MoveL Offs(p0,16.160800000000002,133.0456, 0), v100, z5, tool0;
MoveL Offs(p0,15.9875,133.9125, 0), v100, z5, tool0;
MoveL Offs(p0,15.787200000000002,134.9144, 0), v100, z5, tool0;
MoveL Offs(p0,15.5641,136.0327, 0), v100, z5, tool0;
MoveL Offs(p0,15.322400000000002,137.24880000000002, 0), v100, z5, tool0;
MoveL Offs(p0,15.066300000000002,138.54410000000001, 0), v100, z5, tool0;
MoveL Offs(p0,14.8,139.9, 0), v100, z5, tool0;
MoveL Offs(p0,14.232200000000002,142.5875, 0), v100, z5, tool0;
MoveL Offs(p0,13.713600000000003,144.79200000000006, 0), v100, z5, tool0;
MoveL Offs(p0,13.2214,146.54649999999998, 0), v100, z5, tool0;
MoveL Offs(p0,12.732800000000001,147.88400000000001, 0), v100, z5, tool0;
MoveL Offs(p0,12.225,148.8375, 0), v100, z5, tool0;
MoveL Offs(p0,11.6752,149.44, 0), v100, z5, tool0;
MoveL Offs(p0,11.060599999999999,149.7245, 0), v100, z5, tool0;
MoveL Offs(p0,10.3584,149.72400000000002, 0), v100, z5, tool0;
MoveL Offs(p0,9.5458,149.4715, 0), v100, z5, tool0;
MoveL Offs(p0,8.6,149.0, 0), v100, z5, tool0;
MoveL Offs(p0,8.192600000000002,148.78480000000002, 0), v100, z5, tool0;
MoveL Offs(p0,7.812800000000001,148.56240000000005, 0), v100, z5, tool0;
MoveL Offs(p0,7.4642,148.3376, 0), v100, z5, tool0;
MoveL Offs(p0,7.1504,148.11520000000002, 0), v100, z5, tool0;
MoveL Offs(p0,6.875,147.9, 0), v100, z5, tool0;
MoveL Offs(p0,6.6415999999999995,147.6968, 0), v100, z5, tool0;
MoveL Offs(p0,6.453799999999999,147.51039999999998, 0), v100, z5, tool0;
MoveL Offs(p0,6.3152,147.34560000000002, 0), v100, z5, tool0;
MoveL Offs(p0,6.2294,147.2072, 0), v100, z5, tool0;
MoveL Offs(p0,6.2,147.1, 0), v100, z5, tool0;
MoveL Offs(p0,5.95,144.525, 0), v100, z5, tool0;
MoveL Offs(p0,5.8184,143.6008, 0), v100, z5, tool0;
MoveL Offs(p0,5.6652000000000005,142.57940000000002, 0), v100, z5, tool0;
MoveL Offs(p0,5.492800000000001,141.4776, 0), v100, z5, tool0;
MoveL Offs(p0,5.3036,140.31220000000002, 0), v100, z5, tool0;
MoveL Offs(p0,5.1,139.1, 0), v100, z5, tool0;
MoveL Offs(p0,4.8993,137.8322, 0), v100, z5, tool0;
MoveL Offs(p0,4.718400000000001,136.50560000000002, 0), v100, z5, tool0;
MoveL Offs(p0,4.559099999999999,135.14540000000002, 0), v100, z5, tool0;
MoveL Offs(p0,4.4232000000000005,133.7768, 0), v100, z5, tool0;
MoveL Offs(p0,4.3125,132.425, 0), v100, z5, tool0;
MoveL Offs(p0,4.2288,131.1152, 0), v100, z5, tool0;
MoveL Offs(p0,4.173900000000001,129.8726, 0), v100, z5, tool0;
MoveL Offs(p0,4.1496,128.72240000000002, 0), v100, z5, tool0;
MoveL Offs(p0,4.1577,127.68980000000002, 0), v100, z5, tool0;
MoveL Offs(p0,4.2,126.8, 0), v100, z5, tool0;
MoveL Offs(p0,3.9,123.2, 0), v100, z5, tool0;
MoveL Offs(p0,3.5788,124.12820000000002, 0), v100, z5, tool0;
MoveL Offs(p0,3.334400000000001,125.71760000000003, 0), v100, z5, tool0;
MoveL Offs(p0,3.1656000000000004,127.7954, 0), v100, z5, tool0;
MoveL Offs(p0,3.0712,130.18880000000001, 0), v100, z5, tool0;
MoveL Offs(p0,3.05,132.725, 0), v100, z5, tool0;
MoveL Offs(p0,3.1008,135.2312, 0), v100, z5, tool0;
MoveL Offs(p0,3.2224000000000004,137.5346, 0), v100, z5, tool0;
MoveL Offs(p0,3.4136,139.46240000000003, 0), v100, z5, tool0;
MoveL Offs(p0,3.6732,140.8418, 0), v100, z5, tool0;
MoveL Offs(p0,4.2624,141.74560000000002, 0), v100, z5, tool0;
MoveL Offs(p0,4.3636,141.91039999999998, 0), v100, z5, tool0;
MoveL Offs(p0,4.4432,142.0968, 0), v100, z5, tool0;
MoveL Offs(p0,4.5,142.3, 0), v100, z5, tool0;
MoveL Offs(p0,4.5328,142.5152, 0), v100, z5, tool0;
MoveL Offs(p0,4.5404,142.7376, 0), v100, z5, tool0;
MoveL Offs(p0,4.521600000000001,142.96240000000003, 0), v100, z5, tool0;
MoveL Offs(p0,4.4752,143.18480000000002, 0), v100, z5, tool0;
MoveL Offs(p0,4.4,143.4, 0), v100, z5, tool0;
MoveL Offs(p0,4.9022,146.56709999999998, 0), v100, z5, tool0;
MoveL Offs(p0,5.4144000000000005,148.1312, 0), v100, z5, tool0;
MoveL Offs(p0,6.025,149.7625, 0), v100, z5, tool0;
MoveL Offs(p0,6.6896,151.3488, 0), v100, z5, tool0;
MoveL Offs(p0,7.3638,152.7779, 0), v100, z5, tool0;
MoveL Offs(p0,8.003200000000001,153.93760000000003, 0), v100, z5, tool0;
MoveL Offs(p0,8.563400000000001,154.7157, 0), v100, z5, tool0;
MoveL Offs(p0,9.0,155.0, 0), v100, z5, tool0;
MoveL Offs(p0,9.431999999999999,155.2754, 0), v100, z5, tool0;
MoveL Offs(p0,9.632000000000001,155.4768, 0), v100, z5, tool0;
MoveL Offs(p0,9.85,155.725, 0), v100, z5, tool0;
MoveL Offs(p0,10.080000000000002,156.0152, 0), v100, z5, tool0;
MoveL Offs(p0,10.315999999999999,156.3426, 0), v100, z5, tool0;
MoveL Offs(p0,10.552000000000001,156.7024, 0), v100, z5, tool0;
MoveL Offs(p0,10.782,157.08980000000003, 0), v100, z5, tool0;
MoveL Offs(p0,11.0,157.5, 0), v100, z5, tool0;
MoveL Offs(p0,11.221,157.9102, 0), v100, z5, tool0;
MoveL Offs(p0,11.460000000000004,158.29760000000005, 0), v100, z5, tool0;
MoveL Offs(p0,11.711000000000002,158.6574, 0), v100, z5, tool0;
MoveL Offs(p0,11.968,158.98480000000004, 0), v100, z5, tool0;
MoveL Offs(p0,12.225,159.275, 0), v100, z5, tool0;
MoveL Offs(p0,12.475999999999999,159.5232, 0), v100, z5, tool0;
MoveL Offs(p0,12.715,159.7246, 0), v100, z5, tool0;
MoveL Offs(p0,12.936000000000002,159.8744, 0), v100, z5, tool0;
MoveL Offs(p0,13.133,159.96779999999998, 0), v100, z5, tool0;
MoveL Offs(p0,13.3,160.0, 0), v100, z5, tool0;
MoveL Offs(p0,14.082399999999998,160.29760000000002, 0), v100, z5, tool0;
MoveL Offs(p0,14.3125,160.45, 0), v100, z5, tool0;
MoveL Offs(p0,14.545599999999999,160.62640000000002, 0), v100, z5, tool0;
MoveL Offs(p0,14.7763,160.82319999999999, 0), v100, z5, tool0;
MoveL Offs(p0,14.999200000000002,161.0368, 0), v100, z5, tool0;
MoveL Offs(p0,15.2089,161.2636, 0), v100, z5, tool0;
MoveL Offs(p0,15.4,161.5, 0), v100, z5, tool0;
MoveL Offs(p0,15.943300000000004,162.06070000000003, 0), v100, z5, tool0;
MoveL Offs(p0,16.7584,162.64960000000005, 0), v100, z5, tool0;
MoveL Offs(p0,17.7931,163.24689999999998, 0), v100, z5, tool0;
MoveL Offs(p0,18.995200000000004,163.83280000000002, 0), v100, z5, tool0;
MoveL Offs(p0,20.3125,164.3875, 0), v100, z5, tool0;
MoveL Offs(p0,21.6928,164.8912, 0), v100, z5, tool0;
MoveL Offs(p0,23.0839,165.3241, 0), v100, z5, tool0;
MoveL Offs(p0,24.433600000000006,165.6664, 0), v100, z5, tool0;
MoveL Offs(p0,25.6897,165.8983, 0), v100, z5, tool0;
MoveL Offs(p0,26.8,166.0, 0), v100, z5, tool0;
MoveL Offs(p0,28.5088,165.70880000000002, 0), v100, z5, tool0;
MoveL Offs(p0,28.675,165.4875, 0), v100, z5, tool0;
MoveL Offs(p0,28.7512,165.17919999999998, 0), v100, z5, tool0;
MoveL Offs(p0,28.7446,164.7701, 0), v100, z5, tool0;
MoveL Offs(p0,28.6624,164.2464, 0), v100, z5, tool0;
MoveL Offs(p0,28.5118,163.5943, 0), v100, z5, tool0;
MoveL Offs(p0,28.3,162.8, 0), v100, z5, tool0;
MoveL Offs(p0,28.3,162.8, 0), v100, z5, tool0;
MoveJ Offs(p0,78.0,158.0, 10), v100, z1, tool0;
MoveL Offs(p0,77.6872,153.00560000000004, 0), v100, z5, tool0;
MoveL Offs(p0,77.32230000000001,149.8019, 0), v100, z5, tool0;
MoveL Offs(p0,76.8416,146.2688, 0), v100, z5, tool0;
MoveL Offs(p0,76.2625,142.5125, 0), v100, z5, tool0;
MoveL Offs(p0,75.60239999999999,138.6392, 0), v100, z5, tool0;
MoveL Offs(p0,74.87870000000001,134.7551, 0), v100, z5, tool0;
MoveL Offs(p0,74.1088,130.96640000000002, 0), v100, z5, tool0;
MoveL Offs(p0,73.3101,127.37930000000001, 0), v100, z5, tool0;
MoveL Offs(p0,72.5,124.1, 0), v100, z5, tool0;
MoveL Offs(p0,72.09270000000001,122.5702, 0), v100, z5, tool0;
MoveL Offs(p0,71.71360000000001,121.11360000000005, 0), v100, z5, tool0;
MoveL Offs(p0,71.3669,119.7494, 0), v100, z5, tool0;
MoveL Offs(p0,71.05680000000001,118.49680000000001, 0), v100, z5, tool0;
MoveL Offs(p0,70.7875,117.375, 0), v100, z5, tool0;
MoveL Offs(p0,70.5632,116.4032, 0), v100, z5, tool0;
MoveL Offs(p0,70.3881,115.60059999999999, 0), v100, z5, tool0;
MoveL Offs(p0,70.2664,114.9864, 0), v100, z5, tool0;
MoveL Offs(p0,70.20230000000001,114.5798, 0), v100, z5, tool0;
MoveL Offs(p0,70.2,114.4, 0), v100, z5, tool0;
MoveL Offs(p0,70.48960000000002,114.63760000000002, 0), v100, z5, tool0;
MoveL Offs(p0,70.7499,114.96339999999998, 0), v100, z5, tool0;
MoveL Offs(p0,71.0768,115.41280000000002, 0), v100, z5, tool0;
MoveL Offs(p0,71.4625,115.975, 0), v100, z5, tool0;
MoveL Offs(p0,71.8992,116.6392, 0), v100, z5, tool0;
MoveL Offs(p0,72.3791,117.3946, 0), v100, z5, tool0;
MoveL Offs(p0,72.89440000000002,118.2304, 0), v100, z5, tool0;
MoveL Offs(p0,73.43730000000001,119.13580000000002, 0), v100, z5, tool0;
MoveL Offs(p0,74.0,120.1, 0), v100, z5, tool0;
MoveL Offs(p0,75.3555,122.35350000000001, 0), v100, z5, tool0;
MoveL Offs(p0,76.48000000000003,123.95600000000005, 0), v100, z5, tool0;
MoveL Offs(p0,77.3705,124.9105, 0), v100, z5, tool0;
MoveL Offs(p0,78.024,125.22, 0), v100, z5, tool0;
MoveL Offs(p0,78.4375,124.8875, 0), v100, z5, tool0;
MoveL Offs(p0,78.60800000000002,123.91600000000001, 0), v100, z5, tool0;
MoveL Offs(p0,78.5325,122.30850000000001, 0), v100, z5, tool0;
MoveL Offs(p0,77.6315,117.19750000000002, 0), v100, z5, tool0;
MoveL Offs(p0,76.8,113.7, 0), v100, z5, tool0;
MoveL Offs(p0,75.96640000000001,110.50610000000002, 0), v100, z5, tool0;
MoveL Offs(p0,75.08720000000002,107.46880000000002, 0), v100, z5, tool0;
MoveL Offs(p0,74.16479999999999,104.59470000000002, 0), v100, z5, tool0;
MoveL Offs(p0,73.2016,101.8904, 0), v100, z5, tool0;
MoveL Offs(p0,72.2,99.3625, 0), v100, z5, tool0;
MoveL Offs(p0,71.1624,97.01759999999999, 0), v100, z5, tool0;
MoveL Offs(p0,70.0912,94.8623, 0), v100, z5, tool0;
MoveL Offs(p0,68.9888,92.9032, 0), v100, z5, tool0;
MoveL Offs(p0,67.8576,91.1469, 0), v100, z5, tool0;
MoveL Offs(p0,66.7,89.6, 0), v100, z5, tool0;
MoveL Offs(p0,64.4,86.7, 0), v100, z5, tool0;
MoveL Offs(p0,61.2,92.3, 0), v100, z5, tool0;
MoveL Offs(p0,60.6388,93.25610000000002, 0), v100, z5, tool0;
MoveL Offs(p0,59.9864,94.30880000000003, 0), v100, z5, tool0;
MoveL Offs(p0,59.2596,95.43469999999999, 0), v100, z5, tool0;
MoveL Offs(p0,58.475199999999994,96.6104, 0), v100, z5, tool0;
MoveL Offs(p0,57.65,97.8125, 0), v100, z5, tool0;
MoveL Offs(p0,56.8008,99.01759999999999, 0), v100, z5, tool0;
MoveL Offs(p0,55.944399999999995,100.2023, 0), v100, z5, tool0;
MoveL Offs(p0,55.097600000000014,101.3432, 0), v100, z5, tool0;
MoveL Offs(p0,54.27720000000001,102.41689999999998, 0), v100, z5, tool0;
MoveL Offs(p0,53.5,103.4, 0), v100, z5, tool0;
MoveL Offs(p0,49.0,109.0, 0), v100, z5, tool0;
MoveL Offs(p0,50.9,116.8, 0), v100, z5, tool0;
MoveL Offs(p0,51.2321,118.13260000000002, 0), v100, z5, tool0;
MoveL Offs(p0,51.56480000000001,119.58880000000006, 0), v100, z5, tool0;
MoveL Offs(p0,51.89269999999999,121.13619999999999, 0), v100, z5, tool0;
MoveL Offs(p0,52.21040000000001,122.74240000000002, 0), v100, z5, tool0;
MoveL Offs(p0,52.5125,124.375, 0), v100, z5, tool0;
MoveL Offs(p0,52.793600000000005,126.00160000000001, 0), v100, z5, tool0;
MoveL Offs(p0,53.0483,127.5898, 0), v100, z5, tool0;
MoveL Offs(p0,53.2712,129.1072, 0), v100, z5, tool0;
MoveL Offs(p0,53.4569,130.5214, 0), v100, z5, tool0;
MoveL Offs(p0,53.6,131.8, 0), v100, z5, tool0;
MoveL Offs(p0,53.82320000000002,134.04640000000003, 0), v100, z5, tool0;
MoveL Offs(p0,53.9618,135.0751, 0), v100, z5, tool0;
MoveL Offs(p0,54.113600000000005,136.0192, 0), v100, z5, tool0;
MoveL Offs(p0,54.275,136.8625, 0), v100, z5, tool0;
MoveL Offs(p0,54.4424,137.5888, 0), v100, z5, tool0;
MoveL Offs(p0,54.61220000000001,138.18189999999998, 0), v100, z5, tool0;
MoveL Offs(p0,54.7808,138.62560000000002, 0), v100, z5, tool0;
MoveL Offs(p0,54.9446,138.90370000000001, 0), v100, z5, tool0;
MoveL Offs(p0,55.1,139.0, 0), v100, z5, tool0;
MoveL Offs(p0,55.75040000000003,138.55440000000004, 0), v100, z5, tool0;
MoveL Offs(p0,56.057599999999994,138.03609999999998, 0), v100, z5, tool0;
MoveL Offs(p0,56.34320000000001,137.3552, 0), v100, z5, tool0;
MoveL Offs(p0,56.6,136.5375, 0), v100, z5, tool0;
MoveL Offs(p0,56.8208,135.6088, 0), v100, z5, tool0;
MoveL Offs(p0,56.998400000000004,134.5949, 0), v100, z5, tool0;
MoveL Offs(p0,57.125600000000006,133.5216, 0), v100, z5, tool0;
MoveL Offs(p0,57.1952,132.41469999999998, 0), v100, z5, tool0;
MoveL Offs(p0,57.2,131.3, 0), v100, z5, tool0;
MoveL Offs(p0,57.4403,128.0438, 0), v100, z5, tool0;
MoveL Offs(p0,57.5,128.0, 0), v100, z5, tool0;
MoveL Offs(p0,57.95980000000001,128.5038, 0), v100, z5, tool0;
MoveL Offs(p0,58.43040000000002,129.93040000000002, 0), v100, z5, tool0;
MoveL Offs(p0,58.8986,132.1526, 0), v100, z5, tool0;
MoveL Offs(p0,59.351200000000006,135.0432, 0), v100, z5, tool0;
MoveL Offs(p0,59.775,138.475, 0), v100, z5, tool0;
MoveL Offs(p0,60.15680000000001,142.32080000000002, 0), v100, z5, tool0;
MoveL Offs(p0,60.483399999999996,146.45340000000002, 0), v100, z5, tool0;
MoveL Offs(p0,60.74159999999999,150.74560000000002, 0), v100, z5, tool0;
MoveL Offs(p0,60.9182,155.07020000000003, 0), v100, z5, tool0;
MoveL Offs(p0,61.0,159.3, 0), v100, z5, tool0;
MoveL Offs(p0,61.2125,159.8, 0), v100, z5, tool0;
MoveL Offs(p0,61.30239999999999,159.8688, 0), v100, z5, tool0;
MoveL Offs(p0,61.4067,159.92440000000002, 0), v100, z5, tool0;
MoveL Offs(p0,61.524800000000006,159.9656, 0), v100, z5, tool0;
MoveL Offs(p0,61.6561,159.9912, 0), v100, z5, tool0;
MoveL Offs(p0,61.8,160.0, 0), v100, z5, tool0;
MoveL Offs(p0,62.2879,159.6761, 0), v100, z5, tool0;
MoveL Offs(p0,62.88320000000002,158.78880000000004, 0), v100, z5, tool0;
MoveL Offs(p0,63.54329999999999,157.4647, 0), v100, z5, tool0;
MoveL Offs(p0,64.22560000000001,155.8304, 0), v100, z5, tool0;
MoveL Offs(p0,64.8875,154.0125, 0), v100, z5, tool0;
MoveL Offs(p0,65.4864,152.1376, 0), v100, z5, tool0;
MoveL Offs(p0,65.97970000000001,150.3323, 0), v100, z5, tool0;
MoveL Offs(p0,66.32480000000001,148.7232, 0), v100, z5, tool0;
MoveL Offs(p0,66.47909999999999,147.4369, 0), v100, z5, tool0;
MoveL Offs(p0,66.4,146.6, 0), v100, z5, tool0;
MoveL Offs(p0,65.9839,145.41660000000002, 0), v100, z5, tool0;
MoveL Offs(p0,65.85520000000001,144.77680000000004, 0), v100, z5, tool0;
MoveL Offs(p0,65.9833,144.6362, 0), v100, z5, tool0;
MoveL Offs(p0,66.8875,145.675, 0), v100, z5, tool0;
MoveL Offs(p0,68.4517,148.1778, 0), v100, z5, tool0;
MoveL Offs(p0,69.4048,149.8672, 0), v100, z5, tool0;
MoveL Offs(p0,70.43109999999999,151.7894, 0), v100, z5, tool0;
MoveL Offs(p0,71.5,153.9, 0), v100, z5, tool0;
MoveL Offs(p0,72.72690000000001,156.3719, 0), v100, z5, tool0;
MoveL Offs(p0,73.82720000000003,158.38720000000006, 0), v100, z5, tool0;
MoveL Offs(p0,74.80030000000001,159.9453, 0), v100, z5, tool0;
MoveL Offs(p0,75.64559999999999,161.04560000000004, 0), v100, z5, tool0;
MoveL Offs(p0,76.3625,161.6875, 0), v100, z5, tool0;
MoveL Offs(p0,76.95039999999999,161.8704, 0), v100, z5, tool0;
MoveL Offs(p0,77.4087,161.59369999999998, 0), v100, z5, tool0;
MoveL Offs(p0,77.73679999999999,160.85680000000002, 0), v100, z5, tool0;
MoveL Offs(p0,77.93410000000002,159.65910000000002, 0), v100, z5, tool0;
MoveL Offs(p0,78.0,158.0, 0), v100, z5, tool0;
MoveL Offs(p0,78.0,158.0, 0), v100, z5, tool0;
MoveJ Offs(p0,47.0,140.8, 10), v100, z1, tool0;
MoveL Offs(p0,46.7125,135.0625, 0), v100, z5, tool0;
MoveL Offs(p0,46.5464,134.644, 0), v100, z5, tool0;
MoveL Offs(p0,46.328700000000005,134.40550000000002, 0), v100, z5, tool0;
MoveL Offs(p0,46.052800000000005,134.32000000000002, 0), v100, z5, tool0;
MoveL Offs(p0,45.7121,134.3605, 0), v100, z5, tool0;
MoveL Offs(p0,45.3,134.5, 0), v100, z5, tool0;
MoveL Offs(p0,44.59200000000001,134.71120000000002, 0), v100, z5, tool0;
MoveL Offs(p0,44.1705,134.8348, 0), v100, z5, tool0;
MoveL Offs(p0,43.71600000000001,134.9656, 0), v100, z5, tool0;
MoveL Offs(p0,43.2375,135.1, 0), v100, z5, tool0;
MoveL Offs(p0,42.74399999999999,135.2344, 0), v100, z5, tool0;
MoveL Offs(p0,42.2445,135.36520000000002, 0), v100, z5, tool0;
MoveL Offs(p0,41.748000000000005,135.48880000000003, 0), v100, z5, tool0;
MoveL Offs(p0,41.2635,135.60160000000002, 0), v100, z5, tool0;
MoveL Offs(p0,40.8,135.7, 0), v100, z5, tool0;
MoveL Offs(p0,39.18000000000001,136.12880000000004, 0), v100, z5, tool0;
MoveL Offs(p0,38.64,136.39119999999997, 0), v100, z5, tool0;
MoveL Offs(p0,38.28,136.6824, 0), v100, z5, tool0;
MoveL Offs(p0,38.1,137.0, 0), v100, z5, tool0;
MoveL Offs(p0,38.1,137.3416, 0), v100, z5, tool0;
MoveL Offs(p0,38.279999999999994,137.7048, 0), v100, z5, tool0;
MoveL Offs(p0,38.64,138.0872, 0), v100, z5, tool0;
MoveL Offs(p0,39.18,138.4864, 0), v100, z5, tool0;
MoveL Offs(p0,39.9,138.9, 0), v100, z5, tool0;
MoveL Offs(p0,40.2196,139.13500000000002, 0), v100, z5, tool0;
MoveL Offs(p0,40.57280000000001,139.47200000000004, 0), v100, z5, tool0;
MoveL Offs(p0,40.9512,139.899, 0), v100, z5, tool0;
MoveL Offs(p0,41.3464,140.404, 0), v100, z5, tool0;
MoveL Offs(p0,41.75,140.975, 0), v100, z5, tool0;
MoveL Offs(p0,42.1536,141.6, 0), v100, z5, tool0;
MoveL Offs(p0,42.54880000000001,142.267, 0), v100, z5, tool0;
MoveL Offs(p0,42.927200000000006,142.964, 0), v100, z5, tool0;
MoveL Offs(p0,43.2804,143.679, 0), v100, z5, tool0;
MoveL Offs(p0,43.6,144.4, 0), v100, z5, tool0;
MoveL Offs(p0,43.90500000000001,145.10060000000001, 0), v100, z5, tool0;
MoveL Offs(p0,44.216000000000015,145.75680000000006, 0), v100, z5, tool0;
MoveL Offs(p0,44.527,146.3602, 0), v100, z5, tool0;
MoveL Offs(p0,44.83200000000001,146.9024, 0), v100, z5, tool0;
MoveL Offs(p0,45.125,147.375, 0), v100, z5, tool0;
MoveL Offs(p0,45.4,147.7696, 0), v100, z5, tool0;
MoveL Offs(p0,45.650999999999996,148.0778, 0), v100, z5, tool0;
MoveL Offs(p0,45.872,148.29120000000003, 0), v100, z5, tool0;
MoveL Offs(p0,46.057,148.40140000000002, 0), v100, z5, tool0;
MoveL Offs(p0,46.2,148.4, 0), v100, z5, tool0;
MoveL Offs(p0,46.475200000000015,147.86880000000002, 0), v100, z5, tool0;
MoveL Offs(p0,46.59329999999999,147.3632, 0), v100, z5, tool0;
MoveL Offs(p0,46.6976,146.71840000000003, 0), v100, z5, tool0;
MoveL Offs(p0,46.7875,145.95, 0), v100, z5, tool0;
MoveL Offs(p0,46.862399999999994,145.0736, 0), v100, z5, tool0;
MoveL Offs(p0,46.9217,144.1048, 0), v100, z5, tool0;
MoveL Offs(p0,46.964800000000004,143.0592, 0), v100, z5, tool0;
MoveL Offs(p0,46.9911,141.9524, 0), v100, z5, tool0;
MoveL Offs(p0,47.0,140.8, 0), v100, z5, tool0;
MoveL Offs(p0,47.0,140.8, 0), v100, z5, tool0;
MoveJ Offs(p0,12.0,145.8, 10), v100, z1, tool0;
MoveL Offs(p0,12.342400000000003,144.71920000000006, 0), v100, z5, tool0;
MoveL Offs(p0,12.539100000000001,143.97930000000002, 0), v100, z5, tool0;
MoveL Offs(p0,12.747200000000001,143.12960000000004, 0), v100, z5, tool0;
MoveL Offs(p0,12.9625,142.1875, 0), v100, z5, tool0;
MoveL Offs(p0,13.1808,141.1704, 0), v100, z5, tool0;
MoveL Offs(p0,13.397899999999998,140.0957, 0), v100, z5, tool0;
MoveL Offs(p0,13.6096,138.9808, 0), v100, z5, tool0;
MoveL Offs(p0,13.811700000000002,137.8431, 0), v100, z5, tool0;
MoveL Offs(p0,14.0,136.7, 0), v100, z5, tool0;
MoveL Offs(p0,15.1,130.0, 0), v100, z5, tool0;
MoveL Offs(p0,11.3,125.5, 0), v100, z5, tool0;
MoveL Offs(p0,9.9746,123.9775, 0), v100, z5, tool0;
MoveL Offs(p0,8.868800000000004,122.90800000000004, 0), v100, z5, tool0;
MoveL Offs(p0,7.9682,122.3185, 0), v100, z5, tool0;
MoveL Offs(p0,7.2584,122.23600000000002, 0), v100, z5, tool0;
MoveL Offs(p0,6.725,122.6875, 0), v100, z5, tool0;
MoveL Offs(p0,6.3536,123.7, 0), v100, z5, tool0;
MoveL Offs(p0,6.0392,127.516, 0), v100, z5, tool0;
MoveL Offs(p0,6.067400000000001,130.3735, 0), v100, z5, tool0;
MoveL Offs(p0,6.2,133.9, 0), v100, z5, tool0;
MoveL Offs(p0,6.548000000000002,138.89920000000004, 0), v100, z5, tool0;
MoveL Offs(p0,6.803,141.0028, 0), v100, z5, tool0;
MoveL Offs(p0,7.112,142.8376, 0), v100, z5, tool0;
MoveL Offs(p0,7.475,144.4, 0), v100, z5, tool0;
MoveL Offs(p0,7.892,145.6864, 0), v100, z5, tool0;
MoveL Offs(p0,8.363,146.6932, 0), v100, z5, tool0;
MoveL Offs(p0,8.888000000000002,147.41680000000002, 0), v100, z5, tool0;
MoveL Offs(p0,9.467,147.8536, 0), v100, z5, tool0;
MoveL Offs(p0,10.1,148.0, 0), v100, z5, tool0;
MoveL Offs(p0,10.636399999999998,147.75159999999997, 0), v100, z5, tool0;
MoveL Offs(p0,10.840800000000002,147.57120000000003, 0), v100, z5, tool0;
MoveL Offs(p0,11.05,147.35, 0), v100, z5, tool0;
MoveL Offs(p0,11.259200000000002,147.09279999999998, 0), v100, z5, tool0;
MoveL Offs(p0,11.463600000000001,146.8044, 0), v100, z5, tool0;
MoveL Offs(p0,11.6584,146.48960000000002, 0), v100, z5, tool0;
MoveL Offs(p0,11.8388,146.1532, 0), v100, z5, tool0;
MoveL Offs(p0,12.0,145.8, 0), v100, z5, tool0;
MoveL Offs(p0,12.0,145.8, 0), v100, z5, tool0;
MoveJ Offs(p0,262.7,143.5, 10), v100, z1, tool0;
MoveL Offs(p0,263.8167,142.33740000000003, 0), v100, z5, tool0;
MoveL Offs(p0,264.81760000000014,140.53520000000003, 0), v100, z5, tool0;
MoveL Offs(p0,265.6889,138.19179999999997, 0), v100, z5, tool0;
MoveL Offs(p0,266.4168000000001,135.40560000000002, 0), v100, z5, tool0;
MoveL Offs(p0,266.9875,132.275, 0), v100, z5, tool0;
MoveL Offs(p0,267.3872,128.89839999999998, 0), v100, z5, tool0;
MoveL Offs(p0,267.60209999999995,125.3742, 0), v100, z5, tool0;
MoveL Offs(p0,267.6184,121.80080000000001, 0), v100, z5, tool0;
MoveL Offs(p0,267.4223,118.2766, 0), v100, z5, tool0;
MoveL Offs(p0,267.0,114.9, 0), v100, z5, tool0;
MoveL Offs(p0,265.9941,110.09260000000002, 0), v100, z5, tool0;
MoveL Offs(p0,264.7008000000001,105.73280000000003, 0), v100, z5, tool0;
MoveL Offs(p0,263.0967,101.79419999999998, 0), v100, z5, tool0;
MoveL Offs(p0,261.15840000000003,98.25040000000001, 0), v100, z5, tool0;
MoveL Offs(p0,258.8625,95.075, 0), v100, z5, tool0;
MoveL Offs(p0,256.18559999999997,92.24159999999999, 0), v100, z5, tool0;
MoveL Offs(p0,253.10430000000002,89.7238, 0), v100, z5, tool0;
MoveL Offs(p0,249.59520000000003,87.4952, 0), v100, z5, tool0;
MoveL Offs(p0,245.63490000000002,85.5294, 0), v100, z5, tool0;
MoveL Offs(p0,241.2,83.8, 0), v100, z5, tool0;
MoveL Offs(p0,238.40990000000002,83.00840000000001, 0), v100, z5, tool0;
MoveL Offs(p0,235.25920000000005,82.37520000000002, 0), v100, z5, tool0;
MoveL Offs(p0,231.8373,81.9028, 0), v100, z5, tool0;
MoveL Offs(p0,228.23360000000002,81.59360000000001, 0), v100, z5, tool0;
MoveL Offs(p0,224.5375,81.45, 0), v100, z5, tool0;
MoveL Offs(p0,220.8384,81.4744, 0), v100, z5, tool0;
MoveL Offs(p0,217.22569999999996,81.6692, 0), v100, z5, tool0;
MoveL Offs(p0,213.78879999999998,82.0368, 0), v100, z5, tool0;
MoveL Offs(p0,210.6171,82.5796, 0), v100, z5, tool0;
MoveL Offs(p0,207.8,83.3, 0), v100, z5, tool0;
MoveL Offs(p0,206.86000000000004,83.59630000000001, 0), v100, z5, tool0;
MoveL Offs(p0,205.96800000000002,83.88240000000002, 0), v100, z5, tool0;
MoveL Offs(p0,205.13600000000002,84.1541, 0), v100, z5, tool0;
MoveL Offs(p0,204.376,84.4072, 0), v100, z5, tool0;
MoveL Offs(p0,203.7,84.6375, 0), v100, z5, tool0;
MoveL Offs(p0,203.11999999999998,84.84079999999999, 0), v100, z5, tool0;
MoveL Offs(p0,202.648,85.0129, 0), v100, z5, tool0;
MoveL Offs(p0,202.29600000000002,85.1496, 0), v100, z5, tool0;
MoveL Offs(p0,202.07600000000002,85.2467, 0), v100, z5, tool0;
MoveL Offs(p0,202.0,85.3, 0), v100, z5, tool0;
MoveL Offs(p0,201.7732,86.10370000000002, 0), v100, z5, tool0;
MoveL Offs(p0,201.60640000000004,86.61840000000001, 0), v100, z5, tool0;
MoveL Offs(p0,201.4,87.2375, 0), v100, z5, tool0;
MoveL Offs(p0,201.1576,87.9496, 0), v100, z5, tool0;
MoveL Offs(p0,200.8828,88.7433, 0), v100, z5, tool0;
MoveL Offs(p0,200.57920000000004,89.6072, 0), v100, z5, tool0;
MoveL Offs(p0,200.2504,90.5299, 0), v100, z5, tool0;
MoveL Offs(p0,199.9,91.5, 0), v100, z5, tool0;
MoveL Offs(p0,198.94430000000003,94.961, 0), v100, z5, tool0;
MoveL Offs(p0,198.29040000000006,98.82400000000004, 0), v100, z5, tool0;
MoveL Offs(p0,197.9281,102.939, 0), v100, z5, tool0;
MoveL Offs(p0,197.84720000000002,107.15599999999999, 0), v100, z5, tool0;
MoveL Offs(p0,198.0375,111.325, 0), v100, z5, tool0;
MoveL Offs(p0,198.4888,115.296, 0), v100, z5, tool0;
MoveL Offs(p0,199.1909,118.91900000000001, 0), v100, z5, tool0;
MoveL Offs(p0,200.13360000000003,122.04400000000001, 0), v100, z5, tool0;
MoveL Offs(p0,201.3067,124.521, 0), v100, z5, tool0;
MoveL Offs(p0,202.7,126.2, 0), v100, z5, tool0;
MoveL Offs(p0,203.10110000000003,126.452, 0), v100, z5, tool0;
MoveL Offs(p0,203.65280000000007,126.66800000000003, 0), v100, z5, tool0;
MoveL Offs(p0,204.36769999999999,126.84799999999998, 0), v100, z5, tool0;
MoveL Offs(p0,205.25840000000002,126.992, 0), v100, z5, tool0;
MoveL Offs(p0,206.3375,127.1, 0), v100, z5, tool0;
MoveL Offs(p0,207.61759999999998,127.17199999999998, 0), v100, z5, tool0;
MoveL Offs(p0,209.11129999999997,127.208, 0), v100, z5, tool0;
MoveL Offs(p0,210.8312,127.20800000000001, 0), v100, z5, tool0;
MoveL Offs(p0,212.7899,127.172, 0), v100, z5, tool0;
MoveL Offs(p0,215.0,127.1, 0), v100, z5, tool0;
MoveL Offs(p0,226.12399999999997,127.39519999999997, 0), v100, z5, tool0;
MoveL Offs(p0,227.7715,127.5221, 0), v100, z5, tool0;
MoveL Offs(p0,229.27200000000002,127.66640000000002, 0), v100, z5, tool0;
MoveL Offs(p0,230.59250000000003,127.82629999999999, 0), v100, z5, tool0;
MoveL Offs(p0,231.7,128.0, 0), v100, z5, tool0;
MoveL Offs(p0,234.32330000000002,128.62760000000003, 0), v100, z5, tool0;
MoveL Offs(p0,236.95440000000002,129.42080000000004, 0), v100, z5, tool0;
MoveL Offs(p0,239.56509999999997,130.3652, 0), v100, z5, tool0;
MoveL Offs(p0,242.1272,131.44639999999998, 0), v100, z5, tool0;
MoveL Offs(p0,244.6125,132.65, 0), v100, z5, tool0;
MoveL Offs(p0,246.9928,133.9616, 0), v100, z5, tool0;
MoveL Offs(p0,249.23989999999998,135.36679999999998, 0), v100, z5, tool0;
MoveL Offs(p0,251.32560000000004,136.8512, 0), v100, z5, tool0;
MoveL Offs(p0,253.2217,138.40040000000002, 0), v100, z5, tool0;
MoveL Offs(p0,254.9,140.0, 0), v100, z5, tool0;
MoveL Offs(p0,255.64220000000006,140.7906, 0), v100, z5, tool0;
MoveL Offs(p0,256.36160000000007,141.53680000000006, 0), v100, z5, tool0;
MoveL Offs(p0,257.0474,142.2302, 0), v100, z5, tool0;
MoveL Offs(p0,257.6888,142.86240000000004, 0), v100, z5, tool0;
MoveL Offs(p0,258.275,143.425, 0), v100, z5, tool0;
MoveL Offs(p0,258.79519999999997,143.90959999999998, 0), v100, z5, tool0;
MoveL Offs(p0,259.2386,144.3078, 0), v100, z5, tool0;
MoveL Offs(p0,259.59440000000006,144.6112, 0), v100, z5, tool0;
MoveL Offs(p0,259.8518,144.8114, 0), v100, z5, tool0;
MoveL Offs(p0,260.0,144.9, 0), v100, z5, tool0;
MoveL Offs(p0,260.73440000000005,144.6808, 0), v100, z5, tool0;
MoveL Offs(p0,261.0125,144.5375, 0), v100, z5, tool0;
MoveL Offs(p0,261.31759999999997,144.3672, 0), v100, z5, tool0;
MoveL Offs(p0,261.6443,144.1741, 0), v100, z5, tool0;
MoveL Offs(p0,261.98720000000003,143.9624, 0), v100, z5, tool0;
MoveL Offs(p0,262.34090000000003,143.73630000000003, 0), v100, z5, tool0;
MoveL Offs(p0,262.7,143.5, 0), v100, z5, tool0;
MoveL Offs(p0,262.7,143.5, 0), v100, z5, tool0;
MoveJ Offs(p0,173.4,130.4, 10), v100, z1, tool0;
MoveL Offs(p0,173.71200000000002,120.51520000000002, 0), v100, z5, tool0;
MoveL Offs(p0,173.8875,118.95, 0), v100, z5, tool0;
MoveL Offs(p0,174.11999999999998,117.6128, 0), v100, z5, tool0;
MoveL Offs(p0,174.4185,116.4364, 0), v100, z5, tool0;
MoveL Offs(p0,174.792,115.3536, 0), v100, z5, tool0;
MoveL Offs(p0,175.24949999999998,114.2972, 0), v100, z5, tool0;
MoveL Offs(p0,175.8,113.2, 0), v100, z5, tool0;
MoveL Offs(p0,176.1474,112.48760000000004, 0), v100, z5, tool0;
MoveL Offs(p0,176.46720000000005,111.79680000000003, 0), v100, z5, tool0;
MoveL Offs(p0,176.75579999999997,111.13719999999998, 0), v100, z5, tool0;
MoveL Offs(p0,177.0096,110.51840000000001, 0), v100, z5, tool0;
MoveL Offs(p0,177.225,109.95, 0), v100, z5, tool0;
MoveL Offs(p0,177.3984,109.44160000000002, 0), v100, z5, tool0;
MoveL Offs(p0,177.5262,109.00279999999998, 0), v100, z5, tool0;
MoveL Offs(p0,177.6048,108.64320000000002, 0), v100, z5, tool0;
MoveL Offs(p0,177.63060000000002,108.37240000000001, 0), v100, z5, tool0;
MoveL Offs(p0,177.6,108.2, 0), v100, z5, tool0;
MoveL Offs(p0,177.84660000000002,107.8454, 0), v100, z5, tool0;
MoveL Offs(p0,178.0992,107.7328, 0), v100, z5, tool0;
MoveL Offs(p0,178.425,107.625, 0), v100, z5, tool0;
MoveL Offs(p0,178.8168,107.5232, 0), v100, z5, tool0;
MoveL Offs(p0,179.2674,107.4286, 0), v100, z5, tool0;
MoveL Offs(p0,179.76960000000003,107.3424, 0), v100, z5, tool0;
MoveL Offs(p0,180.3162,107.26579999999998, 0), v100, z5, tool0;
MoveL Offs(p0,180.9,107.2, 0), v100, z5, tool0;
MoveL Offs(p0,184.6,107.0, 0), v100, z5, tool0;
MoveL Offs(p0,185.7,117.7, 0), v100, z5, tool0;
MoveL Offs(p0,186.09040000000005,121.22960000000003, 0), v100, z5, tool0;
MoveL Offs(p0,186.30209999999997,122.9029, 0), v100, z5, tool0;
MoveL Offs(p0,186.5192,124.4808, 0), v100, z5, tool0;
MoveL Offs(p0,186.7375,125.9375, 0), v100, z5, tool0;
MoveL Offs(p0,186.9528,127.24719999999999, 0), v100, z5, tool0;
MoveL Offs(p0,187.1609,128.3841, 0), v100, z5, tool0;
MoveL Offs(p0,187.35760000000002,129.32240000000002, 0), v100, z5, tool0;
MoveL Offs(p0,187.5387,130.0363, 0), v100, z5, tool0;
MoveL Offs(p0,187.7,130.5, 0), v100, z5, tool0;
MoveL Offs(p0,187.9232,131.03990000000005, 0), v100, z5, tool0;
MoveL Offs(p0,188.14160000000007,131.45920000000007, 0), v100, z5, tool0;
MoveL Offs(p0,188.39839999999998,131.75730000000001, 0), v100, z5, tool0;
MoveL Offs(p0,188.73680000000002,131.9336, 0), v100, z5, tool0;
MoveL Offs(p0,189.2,131.9875, 0), v100, z5, tool0;
MoveL Offs(p0,189.8312,131.91840000000002, 0), v100, z5, tool0;
MoveL Offs(p0,190.6736,131.72570000000002, 0), v100, z5, tool0;
MoveL Offs(p0,191.77040000000002,131.4088, 0), v100, z5, tool0;
MoveL Offs(p0,193.1648,130.96710000000002, 0), v100, z5, tool0;
MoveL Offs(p0,196.48150000000004,129.90230000000003, 0), v100, z5, tool0;
MoveL Offs(p0,197.76000000000005,129.47840000000002, 0), v100, z5, tool0;
MoveL Offs(p0,198.7565,129.1121, 0), v100, z5, tool0;
MoveL Offs(p0,199.49200000000002,128.7872, 0), v100, z5, tool0;
MoveL Offs(p0,199.9875,128.4875, 0), v100, z5, tool0;
MoveL Offs(p0,200.26399999999998,128.1968, 0), v100, z5, tool0;
MoveL Offs(p0,200.3425,127.8989, 0), v100, z5, tool0;
MoveL Offs(p0,200.244,127.5776, 0), v100, z5, tool0;
MoveL Offs(p0,199.98950000000002,127.21669999999999, 0), v100, z5, tool0;
MoveL Offs(p0,199.6,126.8, 0), v100, z5, tool0;
MoveL Offs(p0,198.46550000000002,125.1626, 0), v100, z5, tool0;
MoveL Offs(p0,197.47200000000004,122.74880000000003, 0), v100, z5, tool0;
MoveL Offs(p0,196.63449999999997,119.7062, 0), v100, z5, tool0;
MoveL Offs(p0,195.96800000000002,116.18239999999999, 0), v100, z5, tool0;
MoveL Offs(p0,195.4875,112.325, 0), v100, z5, tool0;
MoveL Offs(p0,195.208,108.2816, 0), v100, z5, tool0;
MoveL Offs(p0,195.14449999999997,104.19980000000001, 0), v100, z5, tool0;
MoveL Offs(p0,195.312,100.22720000000001, 0), v100, z5, tool0;
MoveL Offs(p0,195.7255,96.51140000000001, 0), v100, z5, tool0;
MoveL Offs(p0,196.4,93.2, 0), v100, z5, tool0;
MoveL Offs(p0,196.6035,92.34970000000001, 0), v100, z5, tool0;
MoveL Offs(p0,196.79200000000006,91.54560000000002, 0), v100, z5, tool0;
MoveL Offs(p0,196.96249999999998,90.7979, 0), v100, z5, tool0;
MoveL Offs(p0,197.11200000000002,90.11680000000001, 0), v100, z5, tool0;
MoveL Offs(p0,197.2375,89.5125, 0), v100, z5, tool0;
MoveL Offs(p0,197.33599999999998,88.9952, 0), v100, z5, tool0;
MoveL Offs(p0,197.40449999999998,88.57509999999999, 0), v100, z5, tool0;
MoveL Offs(p0,197.44,88.2624, 0), v100, z5, tool0;
MoveL Offs(p0,197.4395,88.0673, 0), v100, z5, tool0;
MoveL Offs(p0,197.4,88.0, 0), v100, z5, tool0;
MoveL Offs(p0,196.17680000000004,88.50400000000003, 0), v100, z5, tool0;
MoveL Offs(p0,195.1977,89.09349999999999, 0), v100, z5, tool0;
MoveL Offs(p0,194.0224,89.87200000000001, 0), v100, z5, tool0;
MoveL Offs(p0,192.6875,90.8125, 0), v100, z5, tool0;
MoveL Offs(p0,191.2296,91.888, 0), v100, z5, tool0;
MoveL Offs(p0,189.68529999999998,93.07149999999999, 0), v100, z5, tool0;
MoveL Offs(p0,188.09120000000001,94.336, 0), v100, z5, tool0;
MoveL Offs(p0,186.4839,95.65450000000001, 0), v100, z5, tool0;
MoveL Offs(p0,184.9,97.0, 0), v100, z5, tool0;
MoveL Offs(p0,183.51500000000004,98.24880000000002, 0), v100, z5, tool0;
MoveL Offs(p0,182.28000000000003,99.44240000000003, 0), v100, z5, tool0;
MoveL Offs(p0,181.16500000000002,100.6216, 0), v100, z5, tool0;
MoveL Offs(p0,180.14000000000004,101.82719999999999, 0), v100, z5, tool0;
MoveL Offs(p0,179.175,103.1, 0), v100, z5, tool0;
MoveL Offs(p0,178.23999999999998,104.4808, 0), v100, z5, tool0;
MoveL Offs(p0,177.305,106.01039999999998, 0), v100, z5, tool0;
MoveL Offs(p0,176.34,107.7296, 0), v100, z5, tool0;
MoveL Offs(p0,175.315,109.6792, 0), v100, z5, tool0;
MoveL Offs(p0,174.2,111.9, 0), v100, z5, tool0;
MoveL Offs(p0,172.95060000000004,114.46790000000001, 0), v100, z5, tool0;
MoveL Offs(p0,171.94480000000004,116.60320000000004, 0), v100, z5, tool0;
MoveL Offs(p0,171.1562,118.4133, 0), v100, z5, tool0;
MoveL Offs(p0,170.5584,120.0056, 0), v100, z5, tool0;
MoveL Offs(p0,170.125,121.4875, 0), v100, z5, tool0;
MoveL Offs(p0,169.8296,122.9664, 0), v100, z5, tool0;
MoveL Offs(p0,169.6458,124.5497, 0), v100, z5, tool0;
MoveL Offs(p0,169.54720000000003,126.3448, 0), v100, z5, tool0;
MoveL Offs(p0,169.50740000000002,128.4591, 0), v100, z5, tool0;
MoveL Offs(p0,169.5,131.0, 0), v100, z5, tool0;
MoveL Offs(p0,169.7052,138.28820000000002, 0), v100, z5, tool0;
MoveL Offs(p0,169.8744,139.9984, 0), v100, z5, tool0;
MoveL Offs(p0,170.1,141.375, 0), v100, z5, tool0;
MoveL Offs(p0,170.3856,142.4336, 0), v100, z5, tool0;
MoveL Offs(p0,170.7348,143.1898, 0), v100, z5, tool0;
MoveL Offs(p0,171.15120000000002,143.6592, 0), v100, z5, tool0;
MoveL Offs(p0,171.6384,143.8574, 0), v100, z5, tool0;
MoveL Offs(p0,172.2,143.8, 0), v100, z5, tool0;
MoveL Offs(p0,172.42800000000003,143.5949, 0), v100, z5, tool0;
MoveL Offs(p0,172.63200000000003,143.15520000000004, 0), v100, z5, tool0;
MoveL Offs(p0,172.81199999999998,142.47430000000003, 0), v100, z5, tool0;
MoveL Offs(p0,172.96800000000002,141.5456, 0), v100, z5, tool0;
MoveL Offs(p0,173.1,140.3625, 0), v100, z5, tool0;
MoveL Offs(p0,173.208,138.9184, 0), v100, z5, tool0;
MoveL Offs(p0,173.292,137.2067, 0), v100, z5, tool0;
MoveL Offs(p0,173.352,135.2208, 0), v100, z5, tool0;
MoveL Offs(p0,173.388,132.9541, 0), v100, z5, tool0;
MoveL Offs(p0,173.4,130.4, 0), v100, z5, tool0;
MoveL Offs(p0,173.4,130.4, 0), v100, z5, tool0;
MoveJ Offs(p0,185.3,127.7, 10), v100, z1, tool0;
MoveL Offs(p0,185.0935,126.62720000000004, 0), v100, z5, tool0;
MoveL Offs(p0,184.89600000000004,125.46560000000004, 0), v100, z5, tool0;
MoveL Offs(p0,184.7105,124.2404, 0), v100, z5, tool0;
MoveL Offs(p0,184.54000000000002,122.9768, 0), v100, z5, tool0;
MoveL Offs(p0,184.3875,121.7, 0), v100, z5, tool0;
MoveL Offs(p0,184.25600000000003,120.43520000000001, 0), v100, z5, tool0;
MoveL Offs(p0,184.14849999999998,119.2076, 0), v100, z5, tool0;
MoveL Offs(p0,184.06800000000004,118.0424, 0), v100, z5, tool0;
MoveL Offs(p0,184.0175,116.96480000000001, 0), v100, z5, tool0;
MoveL Offs(p0,184.0,116.0, 0), v100, z5, tool0;
MoveL Offs(p0,183.7057,111.14000000000001, 0), v100, z5, tool0;
MoveL Offs(p0,183.46240000000003,110.08800000000001, 0), v100, z5, tool0;
MoveL Offs(p0,183.1375,109.3, 0), v100, z5, tool0;
MoveL Offs(p0,182.7256,108.76400000000001, 0), v100, z5, tool0;
MoveL Offs(p0,182.22129999999999,108.468, 0), v100, z5, tool0;
MoveL Offs(p0,181.6192,108.4, 0), v100, z5, tool0;
MoveL Offs(p0,180.9139,108.548, 0), v100, z5, tool0;
MoveL Offs(p0,180.1,108.9, 0), v100, z5, tool0;
MoveL Offs(p0,178.9315,110.03630000000001, 0), v100, z5, tool0;
MoveL Offs(p0,177.84400000000002,112.01440000000002, 0), v100, z5, tool0;
MoveL Offs(p0,176.8645,114.66810000000001, 0), v100, z5, tool0;
MoveL Offs(p0,176.02,117.83120000000001, 0), v100, z5, tool0;
MoveL Offs(p0,175.3375,121.3375, 0), v100, z5, tool0;
MoveL Offs(p0,174.844,125.02080000000001, 0), v100, z5, tool0;
MoveL Offs(p0,174.5665,128.7149, 0), v100, z5, tool0;
MoveL Offs(p0,174.532,132.2536, 0), v100, z5, tool0;
MoveL Offs(p0,174.76749999999998,135.47070000000002, 0), v100, z5, tool0;
MoveL Offs(p0,175.3,138.2, 0), v100, z5, tool0;
MoveL Offs(p0,176.0,141.0, 0), v100, z5, tool0;
MoveL Offs(p0,181.3,137.5, 0), v100, z5, tool0;
MoveL Offs(p0,186.7,133.9, 0), v100, z5, tool0;
MoveL Offs(p0,185.3,127.7, 0), v100, z5, tool0;
MoveL Offs(p0,185.3,127.7, 0), v100, z5, tool0;
MoveJ Offs(p0,45.5,130.0, 10), v100, z1, tool0;
MoveL Offs(p0,50.8,126.9, 0), v100, z5, tool0;
MoveL Offs(p0,48.8,119.7, 0), v100, z5, tool0;
MoveL Offs(p0,48.07540000000001,117.15090000000002, 0), v100, z5, tool0;
MoveL Offs(p0,47.44320000000001,115.05120000000004, 0), v100, z5, tool0;
MoveL Offs(p0,46.8758,113.35230000000001, 0), v100, z5, tool0;
MoveL Offs(p0,46.345600000000005,112.0056, 0), v100, z5, tool0;
MoveL Offs(p0,45.825,110.9625, 0), v100, z5, tool0;
MoveL Offs(p0,45.2864,110.17439999999999, 0), v100, z5, tool0;
MoveL Offs(p0,44.70219999999999,109.5927, 0), v100, z5, tool0;
MoveL Offs(p0,44.0448,109.1688, 0), v100, z5, tool0;
MoveL Offs(p0,43.28660000000001,108.85410000000002, 0), v100, z5, tool0;
MoveL Offs(p0,42.4,108.6, 0), v100, z5, tool0;
MoveL Offs(p0,41.27160000000001,108.23760000000001, 0), v100, z5, tool0;
MoveL Offs(p0,40.0088,107.70480000000005, 0), v100, z5, tool0;
MoveL Offs(p0,38.6452,107.0232, 0), v100, z5, tool0;
MoveL Offs(p0,37.2144,106.2144, 0), v100, z5, tool0;
MoveL Offs(p0,35.75,105.3, 0), v100, z5, tool0;
MoveL Offs(p0,34.2856,104.30160000000001, 0), v100, z5, tool0;
MoveL Offs(p0,32.8548,103.2408, 0), v100, z5, tool0;
MoveL Offs(p0,31.491200000000003,102.1392, 0), v100, z5, tool0;
MoveL Offs(p0,30.2284,101.0184, 0), v100, z5, tool0;
MoveL Offs(p0,29.1,99.9, 0), v100, z5, tool0;
MoveL Offs(p0,26.2,96.9, 0), v100, z5, tool0;
MoveL Offs(p0,23.2,102.2, 0), v100, z5, tool0;
MoveL Offs(p0,22.0104,104.1997, 0), v100, z5, tool0;
MoveL Offs(p0,20.895200000000006,105.94560000000004, 0), v100, z5, tool0;
MoveL Offs(p0,19.8448,107.4479, 0), v100, z5, tool0;
MoveL Offs(p0,18.849600000000002,108.7168, 0), v100, z5, tool0;
MoveL Offs(p0,17.9,109.7625, 0), v100, z5, tool0;
MoveL Offs(p0,16.9864,110.5952, 0), v100, z5, tool0;
MoveL Offs(p0,16.0992,111.2251, 0), v100, z5, tool0;
MoveL Offs(p0,15.228800000000001,111.66240000000002, 0), v100, z5, tool0;
MoveL Offs(p0,14.3656,111.9173, 0), v100, z5, tool0;
MoveL Offs(p0,13.5,112.0, 0), v100, z5, tool0;
MoveL Offs(p0,11.901599999999998,111.7894, 0), v100, z5, tool0;
MoveL Offs(p0,11.583200000000001,111.5488, 0), v100, z5, tool0;
MoveL Offs(p0,11.35,111.175, 0), v100, z5, tool0;
MoveL Offs(p0,11.1888,110.6392, 0), v100, z5, tool0;
MoveL Offs(p0,11.086400000000001,109.9126, 0), v100, z5, tool0;
MoveL Offs(p0,11.029600000000002,108.9664, 0), v100, z5, tool0;
MoveL Offs(p0,11.0052,107.77180000000001, 0), v100, z5, tool0;
MoveL Offs(p0,11.0,106.3, 0), v100, z5, tool0;
MoveL Offs(p0,11.216899999999999,103.1905, 0), v100, z5, tool0;
MoveL Offs(p0,11.340800000000002,102.10800000000002, 0), v100, z5, tool0;
MoveL Offs(p0,11.4875,101.0375, 0), v100, z5, tool0;
MoveL Offs(p0,11.6552,100.0, 0), v100, z5, tool0;
MoveL Offs(p0,11.842099999999999,99.0165, 0), v100, z5, tool0;
MoveL Offs(p0,12.046400000000002,98.108, 0), v100, z5, tool0;
MoveL Offs(p0,12.266300000000001,97.2955, 0), v100, z5, tool0;
MoveL Offs(p0,12.5,96.6, 0), v100, z5, tool0;
MoveL Offs(p0,12.727700000000002,95.94450000000002, 0), v100, z5, tool0;
MoveL Offs(p0,12.929600000000004,95.30400000000003, 0), v100, z5, tool0;
MoveL Offs(p0,13.1039,94.6875, 0), v100, z5, tool0;
MoveL Offs(p0,13.2488,94.10400000000001, 0), v100, z5, tool0;
MoveL Offs(p0,13.3625,93.5625, 0), v100, z5, tool0;
MoveL Offs(p0,13.4432,93.07199999999999, 0), v100, z5, tool0;
MoveL Offs(p0,13.489099999999999,92.6415, 0), v100, z5, tool0;
MoveL Offs(p0,13.498400000000004,92.28000000000002, 0), v100, z5, tool0;
MoveL Offs(p0,13.4693,91.9965, 0), v100, z5, tool0;
MoveL Offs(p0,13.4,91.8, 0), v100, z5, tool0;
MoveL Offs(p0,13.659200000000002,91.0116, 0), v100, z5, tool0;
MoveL Offs(p0,13.8,91.0, 0), v100, z5, tool0;
MoveL Offs(p0,14.363399999999999,90.6301, 0), v100, z5, tool0;
MoveL Offs(p0,14.588800000000003,90.3632, 0), v100, z5, tool0;
MoveL Offs(p0,14.825,90.0375, 0), v100, z5, tool0;
MoveL Offs(p0,15.067200000000003,89.6608, 0), v100, z5, tool0;
MoveL Offs(p0,15.310599999999999,89.24089999999998, 0), v100, z5, tool0;
MoveL Offs(p0,15.550400000000002,88.78560000000002, 0), v100, z5, tool0;
MoveL Offs(p0,15.7818,88.3027, 0), v100, z5, tool0;
MoveL Offs(p0,16.0,87.8, 0), v100, z5, tool0;
MoveL Offs(p0,16.251100000000005,87.24960000000002, 0), v100, z5, tool0;
MoveL Offs(p0,16.5208,86.68480000000002, 0), v100, z5, tool0;
MoveL Offs(p0,16.8037,86.1152, 0), v100, z5, tool0;
MoveL Offs(p0,17.0944,85.5504, 0), v100, z5, tool0;
MoveL Offs(p0,17.3875,85.0, 0), v100, z5, tool0;
MoveL Offs(p0,17.6776,84.4736, 0), v100, z5, tool0;
MoveL Offs(p0,17.9593,83.9808, 0), v100, z5, tool0;
MoveL Offs(p0,18.227200000000003,83.53120000000001, 0), v100, z5, tool0;
MoveL Offs(p0,18.475900000000003,83.1344, 0), v100, z5, tool0;
MoveL Offs(p0,18.7,82.8, 0), v100, z5, tool0;
MoveL Offs(p0,18.930600000000005,82.49860000000001, 0), v100, z5, tool0;
MoveL Offs(p0,19.140800000000006,82.14080000000004, 0), v100, z5, tool0;
MoveL Offs(p0,19.328200000000002,81.7362, 0), v100, z5, tool0;
MoveL Offs(p0,19.4904,81.29440000000001, 0), v100, z5, tool0;
MoveL Offs(p0,19.625,80.825, 0), v100, z5, tool0;
MoveL Offs(p0,19.729599999999998,80.3376, 0), v100, z5, tool0;
MoveL Offs(p0,19.8018,79.84179999999999, 0), v100, z5, tool0;
MoveL Offs(p0,19.839199999999998,79.3472, 0), v100, z5, tool0;
MoveL Offs(p0,19.8394,78.8634, 0), v100, z5, tool0;
MoveL Offs(p0,19.8,78.4, 0), v100, z5, tool0;
MoveL Offs(p0,19.5,75.6, 0), v100, z5, tool0;
MoveL Offs(p0,16.7,79.8, 0), v100, z5, tool0;
MoveL Offs(p0,16.2659,80.51820000000001, 0), v100, z5, tool0;
MoveL Offs(p0,15.867200000000006,81.22560000000001, 0), v100, z5, tool0;
MoveL Offs(p0,15.5093,81.91139999999999, 0), v100, z5, tool0;
MoveL Offs(p0,15.1976,82.5648, 0), v100, z5, tool0;
MoveL Offs(p0,14.9375,83.175, 0), v100, z5, tool0;
MoveL Offs(p0,14.734399999999999,83.73119999999999, 0), v100, z5, tool0;
MoveL Offs(p0,14.593699999999998,84.22259999999999, 0), v100, z5, tool0;
MoveL Offs(p0,14.520800000000003,84.6384, 0), v100, z5, tool0;
MoveL Offs(p0,14.5211,84.9678, 0), v100, z5, tool0;
MoveL Offs(p0,14.6,85.2, 0), v100, z5, tool0;
MoveL Offs(p0,14.825,85.6293, 0), v100, z5, tool0;
MoveL Offs(p0,14.840000000000003,85.72160000000001, 0), v100, z5, tool0;
MoveL Offs(p0,14.825,85.7875, 0), v100, z5, tool0;
MoveL Offs(p0,14.3,85.7, 0), v100, z5, tool0;
MoveL Offs(p0,13.563799999999997,86.25619999999999, 0), v100, z5, tool0;
MoveL Offs(p0,13.2136,86.77040000000001, 0), v100, z5, tool0;
MoveL Offs(p0,12.825,87.425, 0), v100, z5, tool0;
MoveL Offs(p0,12.4064,88.2056, 0), v100, z5, tool0;
MoveL Offs(p0,11.9662,89.09779999999999, 0), v100, z5, tool0;
MoveL Offs(p0,11.512800000000002,90.08720000000001, 0), v100, z5, tool0;
MoveL Offs(p0,11.0546,91.1594, 0), v100, z5, tool0;
MoveL Offs(p0,10.6,92.3, 0), v100, z5, tool0;
MoveL Offs(p0,9.0508,96.8532, 0), v100, z5, tool0;
MoveL Offs(p0,8.058400000000002,101.25760000000004, 0), v100, z5, tool0;
MoveL Offs(p0,7.615599999999999,105.4904, 0), v100, z5, tool0;
MoveL Offs(p0,7.7152,109.5288, 0), v100, z5, tool0;
MoveL Offs(p0,8.35,113.35, 0), v100, z5, tool0;
MoveL Offs(p0,9.512800000000002,116.93119999999999, 0), v100, z5, tool0;
MoveL Offs(p0,11.1964,120.24960000000002, 0), v100, z5, tool0;
MoveL Offs(p0,13.393600000000001,123.28240000000001, 0), v100, z5, tool0;
MoveL Offs(p0,16.097200000000004,126.00680000000003, 0), v100, z5, tool0;
MoveL Offs(p0,19.3,128.4, 0), v100, z5, tool0;
MoveL Offs(p0,21.961400000000005,129.9028, 0), v100, z5, tool0;
MoveL Offs(p0,24.655200000000008,131.11040000000006, 0), v100, z5, tool0;
MoveL Offs(p0,27.365800000000007,132.02159999999998, 0), v100, z5, tool0;
MoveL Offs(p0,30.0776,132.6352, 0), v100, z5, tool0;
MoveL Offs(p0,32.775,132.95, 0), v100, z5, tool0;
MoveL Offs(p0,35.442400000000006,132.9648, 0), v100, z5, tool0;
MoveL Offs(p0,38.06420000000001,132.67839999999998, 0), v100, z5, tool0;
MoveL Offs(p0,40.62480000000001,132.08960000000002, 0), v100, z5, tool0;
MoveL Offs(p0,43.1086,131.1972, 0), v100, z5, tool0;
MoveL Offs(p0,45.5,130.0, 0), v100, z5, tool0;
MoveL Offs(p0,45.5,130.0, 0), v100, z5, tool0;
MoveJ Offs(p0,170.6,110.6, 10), v100, z1, tool0;
MoveL Offs(p0,170.83620000000002,110.0364, 0), v100, z5, tool0;
MoveL Offs(p0,171.00160000000005,109.53520000000003, 0), v100, z5, tool0;
MoveL Offs(p0,171.0914,109.0808, 0), v100, z5, tool0;
MoveL Offs(p0,171.1008,108.6576, 0), v100, z5, tool0;
MoveL Offs(p0,171.025,108.25, 0), v100, z5, tool0;
MoveL Offs(p0,170.85920000000002,107.8424, 0), v100, z5, tool0;
MoveL Offs(p0,170.2384,106.96480000000001, 0), v100, z5, tool0;
MoveL Offs(p0,169.7738,106.4636, 0), v100, z5, tool0;
MoveL Offs(p0,169.2,105.9, 0), v100, z5, tool0;
MoveL Offs(p0,168.74900000000002,105.43500000000002, 0), v100, z5, tool0;
MoveL Offs(p0,168.24400000000006,104.83200000000004, 0), v100, z5, tool0;
MoveL Offs(p0,167.69699999999997,104.109, 0), v100, z5, tool0;
MoveL Offs(p0,167.12,103.28400000000002, 0), v100, z5, tool0;
MoveL Offs(p0,166.525,102.375, 0), v100, z5, tool0;
MoveL Offs(p0,165.92399999999998,101.4, 0), v100, z5, tool0;
MoveL Offs(p0,165.329,100.377, 0), v100, z5, tool0;
MoveL Offs(p0,164.752,99.324, 0), v100, z5, tool0;
MoveL Offs(p0,164.20499999999998,98.259, 0), v100, z5, tool0;
MoveL Offs(p0,163.7,97.2, 0), v100, z5, tool0;
MoveL Offs(p0,162.9874,95.6337, 0), v100, z5, tool0;
MoveL Offs(p0,162.40320000000003,94.25760000000001, 0), v100, z5, tool0;
MoveL Offs(p0,161.9378,93.01589999999999, 0), v100, z5, tool0;
MoveL Offs(p0,161.58160000000004,91.8528, 0), v100, z5, tool0;
MoveL Offs(p0,161.325,90.7125, 0), v100, z5, tool0;
MoveL Offs(p0,161.1584,89.5392, 0), v100, z5, tool0;
MoveL Offs(p0,161.0722,88.27709999999999, 0), v100, z5, tool0;
MoveL Offs(p0,161.0568,86.87039999999999, 0), v100, z5, tool0;
MoveL Offs(p0,161.1026,85.2633, 0), v100, z5, tool0;
MoveL Offs(p0,161.2,83.4, 0), v100, z5, tool0;
MoveL Offs(p0,161.51200000000003,79.4272, 0), v100, z5, tool0;
MoveL Offs(p0,161.74899999999997,77.9298, 0), v100, z5, tool0;
MoveL Offs(p0,162.06400000000002,76.7216, 0), v100, z5, tool0;
MoveL Offs(p0,162.475,75.775, 0), v100, z5, tool0;
MoveL Offs(p0,163.0,75.0624, 0), v100, z5, tool0;
MoveL Offs(p0,163.65699999999998,74.55619999999999, 0), v100, z5, tool0;
MoveL Offs(p0,164.464,74.2288, 0), v100, z5, tool0;
MoveL Offs(p0,165.43900000000002,74.0526, 0), v100, z5, tool0;
MoveL Offs(p0,166.6,74.0, 0), v100, z5, tool0;
MoveL Offs(p0,167.55040000000005,74.30560000000003, 0), v100, z5, tool0;
MoveL Offs(p0,168.1876,74.68039999999999, 0), v100, z5, tool0;
MoveL Offs(p0,168.9232,75.19680000000001, 0), v100, z5, tool0;
MoveL Offs(p0,169.75,75.85, 0), v100, z5, tool0;
MoveL Offs(p0,170.6608,76.63519999999998, 0), v100, z5, tool0;
MoveL Offs(p0,171.64839999999998,77.54759999999999, 0), v100, z5, tool0;
MoveL Offs(p0,172.7056,78.5824, 0), v100, z5, tool0;
MoveL Offs(p0,173.82520000000002,79.7348, 0), v100, z5, tool0;
MoveL Offs(p0,175.0,81.0, 0), v100, z5, tool0;
MoveL Offs(p0,177.6879,83.94640000000001, 0), v100, z5, tool0;
MoveL Offs(p0,179.88320000000004,86.27120000000002, 0), v100, z5, tool0;
MoveL Offs(p0,181.6933,88.0128, 0), v100, z5, tool0;
MoveL Offs(p0,183.22560000000004,89.20960000000001, 0), v100, z5, tool0;
MoveL Offs(p0,184.5875,89.9, 0), v100, z5, tool0;
MoveL Offs(p0,185.8864,90.1224, 0), v100, z5, tool0;
MoveL Offs(p0,187.22969999999998,89.9152, 0), v100, z5, tool0;
MoveL Offs(p0,188.72480000000002,89.31680000000001, 0), v100, z5, tool0;
MoveL Offs(p0,190.47910000000002,88.3656, 0), v100, z5, tool0;
MoveL Offs(p0,192.6,87.1, 0), v100, z5, tool0;
MoveL Offs(p0,199.2,83.1, 0), v100, z5, tool0;
MoveL Offs(p0,195.5,81.6, 0), v100, z5, tool0;
MoveL Offs(p0,194.87730000000002,81.3365, 0), v100, z5, tool0;
MoveL Offs(p0,194.27440000000007,81.08800000000002, 0), v100, z5, tool0;
MoveL Offs(p0,193.6991,80.85749999999999, 0), v100, z5, tool0;
MoveL Offs(p0,193.1592,80.648, 0), v100, z5, tool0;
MoveL Offs(p0,192.6625,80.4625, 0), v100, z5, tool0;
MoveL Offs(p0,192.2168,80.304, 0), v100, z5, tool0;
MoveL Offs(p0,191.8299,80.1755, 0), v100, z5, tool0;
MoveL Offs(p0,191.50960000000003,80.08, 0), v100, z5, tool0;
MoveL Offs(p0,191.26370000000003,80.0205, 0), v100, z5, tool0;
MoveL Offs(p0,191.1,80.0, 0), v100, z5, tool0;
MoveL Offs(p0,190.4762,79.77090000000001, 0), v100, z5, tool0;
MoveL Offs(p0,189.60160000000005,79.12720000000002, 0), v100, z5, tool0;
MoveL Offs(p0,188.5314,78.1343, 0), v100, z5, tool0;
MoveL Offs(p0,187.32080000000002,76.8576, 0), v100, z5, tool0;
MoveL Offs(p0,186.025,75.3625, 0), v100, z5, tool0;
MoveL Offs(p0,184.6992,73.7144, 0), v100, z5, tool0;
MoveL Offs(p0,183.3986,71.9787, 0), v100, z5, tool0;
MoveL Offs(p0,182.1784,70.22080000000001, 0), v100, z5, tool0;
MoveL Offs(p0,181.09380000000002,68.5061, 0), v100, z5, tool0;
MoveL Offs(p0,180.2,66.9, 0), v100, z5, tool0;
MoveL Offs(p0,179.5384,65.56150000000001, 0), v100, z5, tool0;
MoveL Offs(p0,178.98720000000006,64.34000000000002, 0), v100, z5, tool0;
MoveL Offs(p0,178.5368,63.1965, 0), v100, z5, tool0;
MoveL Offs(p0,178.1776,62.092000000000006, 0), v100, z5, tool0;
MoveL Offs(p0,177.9,60.9875, 0), v100, z5, tool0;
MoveL Offs(p0,177.6944,59.84400000000001, 0), v100, z5, tool0;
MoveL Offs(p0,177.5512,58.62249999999999, 0), v100, z5, tool0;
MoveL Offs(p0,177.4608,57.284000000000006, 0), v100, z5, tool0;
MoveL Offs(p0,177.4136,55.7895, 0), v100, z5, tool0;
MoveL Offs(p0,177.4,54.1, 0), v100, z5, tool0;
MoveL Offs(p0,177.1264,48.37599999999999, 0), v100, z5, tool0;
MoveL Offs(p0,177.01219999999998,47.796499999999995, 0), v100, z5, tool0;
MoveL Offs(p0,176.88479999999998,47.364, 0), v100, z5, tool0;
MoveL Offs(p0,176.7466,47.093500000000006, 0), v100, z5, tool0;
MoveL Offs(p0,176.6,47.0, 0), v100, z5, tool0;
MoveL Offs(p0,176.00320000000005,47.273600000000016, 0), v100, z5, tool0;
MoveL Offs(p0,175.54429999999996,47.5994, 0), v100, z5, tool0;
MoveL Offs(p0,174.99360000000001,48.0368, 0), v100, z5, tool0;
MoveL Offs(p0,174.3625,48.575, 0), v100, z5, tool0;
MoveL Offs(p0,173.6624,49.2032, 0), v100, z5, tool0;
MoveL Offs(p0,172.9047,49.9106, 0), v100, z5, tool0;
MoveL Offs(p0,172.10080000000002,50.686400000000006, 0), v100, z5, tool0;
MoveL Offs(p0,171.2621,51.5198, 0), v100, z5, tool0;
MoveL Offs(p0,170.4,52.4, 0), v100, z5, tool0;
MoveL Offs(p0,168.71130000000002,54.21390000000001, 0), v100, z5, tool0;
MoveL Offs(p0,167.12640000000005,56.11120000000002, 0), v100, z5, tool0;
MoveL Offs(p0,165.64709999999997,58.0853, 0), v100, z5, tool0;
MoveL Offs(p0,164.27519999999998,60.1296, 0), v100, z5, tool0;
MoveL Offs(p0,163.0125,62.2375, 0), v100, z5, tool0;
MoveL Offs(p0,161.8608,64.4024, 0), v100, z5, tool0;
MoveL Offs(p0,160.82189999999997,66.6177, 0), v100, z5, tool0;
MoveL Offs(p0,159.8976,68.8768, 0), v100, z5, tool0;
MoveL Offs(p0,159.0897,71.1731, 0), v100, z5, tool0;
MoveL Offs(p0,158.4,73.5, 0), v100, z5, tool0;
MoveL Offs(p0,157.98370000000003,75.4732, 0), v100, z5, tool0;
MoveL Offs(p0,157.63760000000005,77.92160000000003, 0), v100, z5, tool0;
MoveL Offs(p0,157.3659,80.6784, 0), v100, z5, tool0;
MoveL Offs(p0,157.1728,83.5768, 0), v100, z5, tool0;
MoveL Offs(p0,157.0625,86.45, 0), v100, z5, tool0;
MoveL Offs(p0,157.03920000000002,89.1312, 0), v100, z5, tool0;
MoveL Offs(p0,157.1071,91.45360000000001, 0), v100, z5, tool0;
MoveL Offs(p0,157.27040000000002,93.25040000000001, 0), v100, z5, tool0;
MoveL Offs(p0,157.5333,94.35480000000001, 0), v100, z5, tool0;
MoveL Offs(p0,157.9,94.6, 0), v100, z5, tool0;
MoveL Offs(p0,158.4328,94.852, 0), v100, z5, tool0;
MoveL Offs(p0,158.4404,95.05850000000001, 0), v100, z5, tool0;
MoveL Offs(p0,158.4216,95.304, 0), v100, z5, tool0;
MoveL Offs(p0,158.3752,95.5855, 0), v100, z5, tool0;
MoveL Offs(p0,158.3,95.9, 0), v100, z5, tool0;
MoveL Offs(p0,158.6125,98.4, 0), v100, z5, tool0;
MoveL Offs(p0,158.804,99.0608, 0), v100, z5, tool0;
MoveL Offs(p0,159.0315,99.7444, 0), v100, z5, tool0;
MoveL Offs(p0,159.292,100.4376, 0), v100, z5, tool0;
MoveL Offs(p0,159.5825,101.1272, 0), v100, z5, tool0;
MoveL Offs(p0,159.9,101.8, 0), v100, z5, tool0;
MoveL Offs(p0,160.62990000000002,103.13420000000004, 0), v100, z5, tool0;
MoveL Offs(p0,161.52720000000005,104.57760000000003, 0), v100, z5, tool0;
MoveL Offs(p0,162.5433,106.0714, 0), v100, z5, tool0;
MoveL Offs(p0,163.6296,107.5568, 0), v100, z5, tool0;
MoveL Offs(p0,164.7375,108.975, 0), v100, z5, tool0;
MoveL Offs(p0,165.81839999999997,110.2672, 0), v100, z5, tool0;
MoveL Offs(p0,166.8237,111.37460000000002, 0), v100, z5, tool0;
MoveL Offs(p0,167.70480000000003,112.2384, 0), v100, z5, tool0;
MoveL Offs(p0,168.41310000000001,112.7998, 0), v100, z5, tool0;
MoveL Offs(p0,168.9,113.0, 0), v100, z5, tool0;
MoveL Offs(p0,169.2861,112.72729999999999, 0), v100, z5, tool0;
MoveL Offs(p0,169.45520000000002,112.52960000000003, 0), v100, z5, tool0;
MoveL Offs(p0,169.6375,112.2875, 0), v100, z5, tool0;
MoveL Offs(p0,169.8288,112.00640000000001, 0), v100, z5, tool0;
MoveL Offs(p0,170.0249,111.6917, 0), v100, z5, tool0;
MoveL Offs(p0,170.22160000000002,111.34880000000003, 0), v100, z5, tool0;
MoveL Offs(p0,170.4147,110.98310000000001, 0), v100, z5, tool0;
MoveL Offs(p0,170.6,110.6, 0), v100, z5, tool0;
MoveL Offs(p0,170.6,110.6, 0), v100, z5, tool0;
MoveJ Offs(p0,18.8,106.1, 10), v100, z1, tool0;
MoveL Offs(p0,20.518600000000003,103.89590000000001, 0), v100, z5, tool0;
MoveL Offs(p0,21.904800000000005,101.97920000000002, 0), v100, z5, tool0;
MoveL Offs(p0,22.9742,100.28329999999998, 0), v100, z5, tool0;
MoveL Offs(p0,23.742400000000004,98.7416, 0), v100, z5, tool0;
MoveL Offs(p0,24.225,97.2875, 0), v100, z5, tool0;
MoveL Offs(p0,24.4376,95.8544, 0), v100, z5, tool0;
MoveL Offs(p0,24.3958,94.37570000000001, 0), v100, z5, tool0;
MoveL Offs(p0,24.115200000000005,92.78480000000002, 0), v100, z5, tool0;
MoveL Offs(p0,23.611400000000003,91.0151, 0), v100, z5, tool0;
MoveL Offs(p0,22.9,89.0, 0), v100, z5, tool0;
MoveL Offs(p0,20.7,82.8, 0), v100, z5, tool0;
MoveL Offs(p0,18.3,86.7, 0), v100, z5, tool0;
MoveL Offs(p0,16.8345,89.39730000000002, 0), v100, z5, tool0;
MoveL Offs(p0,15.516000000000005,92.41440000000003, 0), v100, z5, tool0;
MoveL Offs(p0,14.371500000000001,95.60909999999998, 0), v100, z5, tool0;
MoveL Offs(p0,13.428,98.8392, 0), v100, z5, tool0;
MoveL Offs(p0,12.7125,101.9625, 0), v100, z5, tool0;
MoveL Offs(p0,12.251999999999999,104.8368, 0), v100, z5, tool0;
MoveL Offs(p0,12.0735,107.3199, 0), v100, z5, tool0;
MoveL Offs(p0,12.204000000000002,109.26960000000001, 0), v100, z5, tool0;
MoveL Offs(p0,12.6705,110.54369999999999, 0), v100, z5, tool0;
MoveL Offs(p0,13.5,111.0, 0), v100, z5, tool0;
MoveL Offs(p0,14.156800000000004,110.74960000000003, 0), v100, z5, tool0;
MoveL Offs(p0,14.6007,110.45189999999998, 0), v100, z5, tool0;
MoveL Offs(p0,15.106400000000002,110.0528, 0), v100, z5, tool0;
MoveL Offs(p0,15.6625,109.5625, 0), v100, z5, tool0;
MoveL Offs(p0,16.257600000000004,108.9912, 0), v100, z5, tool0;
MoveL Offs(p0,16.8803,108.34909999999999, 0), v100, z5, tool0;
MoveL Offs(p0,17.5192,107.6464, 0), v100, z5, tool0;
MoveL Offs(p0,18.1629,106.8933, 0), v100, z5, tool0;
MoveL Offs(p0,18.8,106.1, 0), v100, z5, tool0;
MoveL Offs(p0,18.8,106.1, 0), v100, z5, tool0;
MoveJ Offs(p0,51.2,100.8, 10), v100, z1, tool0;
MoveL Offs(p0,52.76220000000001,99.0823, 0), v100, z5, tool0;
MoveL Offs(p0,54.145600000000016,97.47440000000002, 0), v100, z5, tool0;
MoveL Offs(p0,55.345400000000005,95.98409999999998, 0), v100, z5, tool0;
MoveL Offs(p0,56.35680000000001,94.6192, 0), v100, z5, tool0;
MoveL Offs(p0,57.175,93.3875, 0), v100, z5, tool0;
MoveL Offs(p0,57.7952,92.2968, 0), v100, z5, tool0;
MoveL Offs(p0,58.212599999999995,91.3549, 0), v100, z5, tool0;
MoveL Offs(p0,58.42240000000002,90.56960000000001, 0), v100, z5, tool0;
MoveL Offs(p0,58.41980000000001,89.9487, 0), v100, z5, tool0;
MoveL Offs(p0,58.2,89.5, 0), v100, z5, tool0;
MoveL Offs(p0,57.9966,89.1796, 0), v100, z5, tool0;
MoveL Offs(p0,57.99520000000001,89.1272, 0), v100, z5, tool0;
MoveL Offs(p0,58.4322,89.2192, 0), v100, z5, tool0;
MoveL Offs(p0,58.6,89.3, 0), v100, z5, tool0;
MoveL Offs(p0,59.36480000000002,89.05040000000002, 0), v100, z5, tool0;
MoveL Offs(p0,59.8582,88.59710000000001, 0), v100, z5, tool0;
MoveL Offs(p0,60.3744,87.9992, 0), v100, z5, tool0;
MoveL Offs(p0,60.875,87.3125, 0), v100, z5, tool0;
MoveL Offs(p0,61.32159999999999,86.5928, 0), v100, z5, tool0;
MoveL Offs(p0,61.6758,85.89590000000001, 0), v100, z5, tool0;
MoveL Offs(p0,61.89919999999999,85.2776, 0), v100, z5, tool0;
MoveL Offs(p0,61.9534,84.79370000000002, 0), v100, z5, tool0;
MoveL Offs(p0,61.8,84.5, 0), v100, z5, tool0;
MoveL Offs(p0,60.4147,83.52580000000002, 0), v100, z5, tool0;
MoveL Offs(p0,59.14160000000002,82.58640000000003, 0), v100, z5, tool0;
MoveL Offs(p0,57.9849,81.6866, 0), v100, z5, tool0;
MoveL Offs(p0,56.948800000000006,80.83120000000001, 0), v100, z5, tool0;
MoveL Offs(p0,56.0375,80.025, 0), v100, z5, tool0;
MoveL Offs(p0,55.2552,79.27279999999999, 0), v100, z5, tool0;
MoveL Offs(p0,54.60609999999999,78.57939999999999, 0), v100, z5, tool0;
MoveL Offs(p0,54.09440000000001,77.9496, 0), v100, z5, tool0;
MoveL Offs(p0,53.72429999999999,77.38820000000001, 0), v100, z5, tool0;
MoveL Offs(p0,53.5,76.9, 0), v100, z5, tool0;
MoveL Offs(p0,53.22720000000002,76.31840000000003, 0), v100, z5, tool0;
MoveL Offs(p0,53.0698,76.0486, 0), v100, z5, tool0;
MoveL Offs(p0,52.90160000000001,75.79920000000001, 0), v100, z5, tool0;
MoveL Offs(p0,52.725,75.575, 0), v100, z5, tool0;
MoveL Offs(p0,52.5424,75.3808, 0), v100, z5, tool0;
MoveL Offs(p0,52.35619999999999,75.22139999999999, 0), v100, z5, tool0;
MoveL Offs(p0,52.16880000000001,75.1016, 0), v100, z5, tool0;
MoveL Offs(p0,51.982600000000005,75.0262, 0), v100, z5, tool0;
MoveL Offs(p0,51.8,75.0, 0), v100, z5, tool0;
MoveL Offs(p0,50.390400000000014,75.59920000000002, 0), v100, z5, tool0;
MoveL Offs(p0,49.4501,76.25280000000001, 0), v100, z5, tool0;
MoveL Offs(p0,48.443200000000004,77.05760000000001, 0), v100, z5, tool0;
MoveL Offs(p0,47.4375,77.95, 0), v100, z5, tool0;
MoveL Offs(p0,46.5008,78.8664, 0), v100, z5, tool0;
MoveL Offs(p0,45.7009,79.7432, 0), v100, z5, tool0;
MoveL Offs(p0,45.1056,80.51680000000002, 0), v100, z5, tool0;
MoveL Offs(p0,44.7827,81.12360000000001, 0), v100, z5, tool0;
MoveL Offs(p0,44.8,81.5, 0), v100, z5, tool0;
MoveL Offs(p0,45.006099999999996,81.8033, 0), v100, z5, tool0;
MoveL Offs(p0,45.0112,81.8776, 0), v100, z5, tool0;
MoveL Offs(p0,44.5,82.0, 0), v100, z5, tool0;
MoveL Offs(p0,41.483,82.3955, 0), v100, z5, tool0;
MoveL Offs(p0,41.412,82.656, 0), v100, z5, tool0;
MoveL Offs(p0,41.449,82.9585, 0), v100, z5, tool0;
MoveL Offs(p0,41.6,83.3, 0), v100, z5, tool0;
MoveL Offs(p0,41.84929999999999,83.7482, 0), v100, z5, tool0;
MoveL Offs(p0,41.881600000000006,83.85040000000001, 0), v100, z5, tool0;
MoveL Offs(p0,41.8875,83.925, 0), v100, z5, tool0;
MoveL Offs(p0,41.8664,83.96959999999999, 0), v100, z5, tool0;
MoveL Offs(p0,41.8177,83.98179999999999, 0), v100, z5, tool0;
MoveL Offs(p0,39.324,84.08160000000001, 0), v100, z5, tool0;
MoveL Offs(p0,38.962,84.27520000000001, 0), v100, z5, tool0;
MoveL Offs(p0,38.6,84.5, 0), v100, z5, tool0;
MoveL Offs(p0,37.746300000000005,85.013, 0), v100, z5, tool0;
MoveL Offs(p0,36.8224,85.41200000000002, 0), v100, z5, tool0;
MoveL Offs(p0,35.8541,85.697, 0), v100, z5, tool0;
MoveL Offs(p0,34.8672,85.86800000000001, 0), v100, z5, tool0;
MoveL Offs(p0,33.8875,85.925, 0), v100, z5, tool0;
MoveL Offs(p0,32.940799999999996,85.868, 0), v100, z5, tool0;
MoveL Offs(p0,32.0529,85.697, 0), v100, z5, tool0;
MoveL Offs(p0,31.249599999999997,85.412, 0), v100, z5, tool0;
MoveL Offs(p0,30.5567,85.013, 0), v100, z5, tool0;
MoveL Offs(p0,29.293200000000002,83.04100000000001, 0), v100, z5, tool0;
MoveL Offs(p0,29.121600000000008,81.07200000000003, 0), v100, z5, tool0;
MoveL Offs(p0,29.4384,78.69500000000001, 0), v100, z5, tool0;
MoveL Offs(p0,31.35,73.125, 0), v100, z5, tool0;
MoveL Offs(p0,32.8512,70.136, 0), v100, z5, tool0;
MoveL Offs(p0,34.653600000000004,67.147, 0), v100, z5, tool0;
MoveL Offs(p0,36.71040000000001,64.26000000000002, 0), v100, z5, tool0;
MoveL Offs(p0,38.9748,61.577, 0), v100, z5, tool0;
MoveL Offs(p0,41.4,59.2, 0), v100, z5, tool0;
MoveL Offs(p0,42.33300000000001,58.356700000000004, 0), v100, z5, tool0;
MoveL Offs(p0,43.10400000000001,57.601600000000005, 0), v100, z5, tool0;
MoveL Offs(p0,43.730999999999995,56.896899999999995, 0), v100, z5, tool0;
MoveL Offs(p0,44.23200000000001,56.20480000000001, 0), v100, z5, tool0;
MoveL Offs(p0,44.625,55.4875, 0), v100, z5, tool0;
MoveL Offs(p0,44.928000000000004,54.7072, 0), v100, z5, tool0;
MoveL Offs(p0,45.159000000000006,53.8261, 0), v100, z5, tool0;
MoveL Offs(p0,45.336,52.80640000000001, 0), v100, z5, tool0;
MoveL Offs(p0,45.477,51.61030000000001, 0), v100, z5, tool0;
MoveL Offs(p0,45.6,50.2, 0), v100, z5, tool0;
MoveL Offs(p0,45.8475,47.4235, 0), v100, z5, tool0;
MoveL Offs(p0,45.952000000000005,46.544, 0), v100, z5, tool0;
MoveL Offs(p0,46.0625,45.7125, 0), v100, z5, tool0;
MoveL Offs(p0,46.176,44.944, 0), v100, z5, tool0;
MoveL Offs(p0,46.2895,44.2535, 0), v100, z5, tool0;
MoveL Offs(p0,46.400000000000006,43.656000000000006, 0), v100, z5, tool0;
MoveL Offs(p0,46.5045,43.1665, 0), v100, z5, tool0;
MoveL Offs(p0,46.6,42.8, 0), v100, z5, tool0;
MoveL Offs(p0,46.2679,41.0234, 0), v100, z5, tool0;
MoveL Offs(p0,46.1,41.0, 0), v100, z5, tool0;
MoveL Offs(p0,45.3624,41.244800000000005, 0), v100, z5, tool0;
MoveL Offs(p0,44.243200000000016,41.914400000000015, 0), v100, z5, tool0;
MoveL Offs(p0,42.852799999999995,42.91159999999999, 0), v100, z5, tool0;
MoveL Offs(p0,41.3016,44.1392, 0), v100, z5, tool0;
MoveL Offs(p0,39.7,45.5, 0), v100, z5, tool0;
MoveL Offs(p0,38.15839999999999,46.896800000000006, 0), v100, z5, tool0;
MoveL Offs(p0,36.7872,48.2324, 0), v100, z5, tool0;
MoveL Offs(p0,35.6968,49.409600000000005, 0), v100, z5, tool0;
MoveL Offs(p0,34.9976,50.3312, 0), v100, z5, tool0;
MoveL Offs(p0,34.8,50.9, 0), v100, z5, tool0;
MoveL Offs(p0,34.5912,51.663199999999996, 0), v100, z5, tool0;
MoveL Offs(p0,34.4906,51.67909999999999, 0), v100, z5, tool0;
MoveL Offs(p0,34.3744,51.65840000000001, 0), v100, z5, tool0;
MoveL Offs(p0,34.2438,51.59930000000001, 0), v100, z5, tool0;
MoveL Offs(p0,34.1,51.5, 0), v100, z5, tool0;
MoveL Offs(p0,32.92720000000001,51.907200000000024, 0), v100, z5, tool0;
MoveL Offs(p0,32.135299999999994,52.7078, 0), v100, z5, tool0;
MoveL Offs(p0,31.245600000000003,53.84560000000001, 0), v100, z5, tool0;
MoveL Offs(p0,30.2875,55.275, 0), v100, z5, tool0;
MoveL Offs(p0,29.290399999999998,56.9504, 0), v100, z5, tool0;
MoveL Offs(p0,28.2837,58.82620000000001, 0), v100, z5, tool0;
MoveL Offs(p0,27.2968,60.8568, 0), v100, z5, tool0;
MoveL Offs(p0,26.3591,62.9966, 0), v100, z5, tool0;
MoveL Offs(p0,25.5,65.2, 0), v100, z5, tool0;
MoveL Offs(p0,24.6991,67.6564, 0), v100, z5, tool0;
MoveL Offs(p0,24.096800000000005,70.0552, 0), v100, z5, tool0;
MoveL Offs(p0,23.6937,72.41080000000001, 0), v100, z5, tool0;
MoveL Offs(p0,23.4904,74.7376, 0), v100, z5, tool0;
MoveL Offs(p0,23.4875,77.05, 0), v100, z5, tool0;
MoveL Offs(p0,23.6856,79.36240000000001, 0), v100, z5, tool0;
MoveL Offs(p0,24.0853,81.6892, 0), v100, z5, tool0;
MoveL Offs(p0,24.6872,84.04480000000001, 0), v100, z5, tool0;
MoveL Offs(p0,26.5,88.9, 0), v100, z5, tool0;
MoveL Offs(p0,27.755500000000005,91.3147, 0), v100, z5, tool0;
MoveL Offs(p0,29.32000000000001,93.72160000000004, 0), v100, z5, tool0;
MoveL Offs(p0,31.1305,96.0649, 0), v100, z5, tool0;
MoveL Offs(p0,33.124,98.28880000000001, 0), v100, z5, tool0;
MoveL Offs(p0,35.2375,100.3375, 0), v100, z5, tool0;
MoveL Offs(p0,37.408,102.15520000000001, 0), v100, z5, tool0;
MoveL Offs(p0,39.572500000000005,103.68610000000001, 0), v100, z5, tool0;
MoveL Offs(p0,41.668000000000006,104.87440000000001, 0), v100, z5, tool0;
MoveL Offs(p0,43.6315,105.6643, 0), v100, z5, tool0;
MoveL Offs(p0,45.4,106.0, 0), v100, z5, tool0;
MoveL Offs(p0,45.936000000000014,105.72800000000004, 0), v100, z5, tool0;
MoveL Offs(p0,46.363,105.40600000000002, 0), v100, z5, tool0;
MoveL Offs(p0,46.88,104.97600000000003, 0), v100, z5, tool0;
MoveL Offs(p0,47.475,104.45, 0), v100, z5, tool0;
MoveL Offs(p0,48.135999999999996,103.84, 0), v100, z5, tool0;
MoveL Offs(p0,48.851,103.15799999999999, 0), v100, z5, tool0;
MoveL Offs(p0,49.608000000000004,102.41600000000001, 0), v100, z5, tool0;
MoveL Offs(p0,50.395,101.626, 0), v100, z5, tool0;
MoveL Offs(p0,51.2,100.8, 0), v100, z5, tool0;
MoveL Offs(p0,51.2,100.8, 0), v100, z5, tool0;
MoveJ Offs(p0,174.0,105.2, 10), v100, z1, tool0;
MoveL Offs(p0,174.26160000000004,104.66720000000002, 0), v100, z5, tool0;
MoveL Offs(p0,174.5724,104.2028, 0), v100, z5, tool0;
MoveL Offs(p0,174.98880000000003,103.6256, 0), v100, z5, tool0;
MoveL Offs(p0,175.5,102.95, 0), v100, z5, tool0;
MoveL Offs(p0,176.0952,102.1904, 0), v100, z5, tool0;
MoveL Offs(p0,176.7636,101.3612, 0), v100, z5, tool0;
MoveL Offs(p0,177.49439999999998,100.4768, 0), v100, z5, tool0;
MoveL Offs(p0,178.2768,99.55160000000001, 0), v100, z5, tool0;
MoveL Offs(p0,179.1,98.6, 0), v100, z5, tool0;
MoveL Offs(p0,184.3,92.8, 0), v100, z5, tool0;
MoveL Offs(p0,175.9,84.4, 0), v100, z5, tool0;
MoveL Offs(p0,174.52650000000003,83.047, 0), v100, z5, tool0;
MoveL Offs(p0,173.18000000000006,81.76000000000002, 0), v100, z5, tool0;
MoveL Offs(p0,171.88150000000002,80.55699999999999, 0), v100, z5, tool0;
MoveL Offs(p0,170.652,79.45599999999999, 0), v100, z5, tool0;
MoveL Offs(p0,169.5125,78.475, 0), v100, z5, tool0;
MoveL Offs(p0,168.484,77.63199999999999, 0), v100, z5, tool0;
MoveL Offs(p0,167.5875,76.94500000000001, 0), v100, z5, tool0;
MoveL Offs(p0,166.844,76.43200000000002, 0), v100, z5, tool0;
MoveL Offs(p0,166.2745,76.111, 0), v100, z5, tool0;
MoveL Offs(p0,165.9,76.0, 0), v100, z5, tool0;
MoveL Offs(p0,164.49169999999998,76.5454, 0), v100, z5, tool0;
MoveL Offs(p0,163.54960000000005,78.05920000000003, 0), v100, z5, tool0;
MoveL Offs(p0,163.04789999999997,80.3578, 0), v100, z5, tool0;
MoveL Offs(p0,162.9608,83.2576, 0), v100, z5, tool0;
MoveL Offs(p0,163.2625,86.575, 0), v100, z5, tool0;
MoveL Offs(p0,163.9272,90.1264, 0), v100, z5, tool0;
MoveL Offs(p0,164.9291,93.7282, 0), v100, z5, tool0;
MoveL Offs(p0,166.24240000000003,97.19680000000001, 0), v100, z5, tool0;
MoveL Offs(p0,167.8413,100.3486, 0), v100, z5, tool0;
MoveL Offs(p0,169.7,103.0, 0), v100, z5, tool0;
MoveL Offs(p0,170.4036,103.8122, 0), v100, z5, tool0;
MoveL Offs(p0,171.06880000000007,104.50560000000003, 0), v100, z5, tool0;
MoveL Offs(p0,171.68720000000002,105.07540000000002, 0), v100, z5, tool0;
MoveL Offs(p0,172.25040000000004,105.51680000000002, 0), v100, z5, tool0;
MoveL Offs(p0,172.75,105.825, 0), v100, z5, tool0;
MoveL Offs(p0,173.17759999999998,105.9952, 0), v100, z5, tool0;
MoveL Offs(p0,173.5248,106.02259999999998, 0), v100, z5, tool0;
MoveL Offs(p0,173.78320000000002,105.90240000000001, 0), v100, z5, tool0;
MoveL Offs(p0,173.94440000000003,105.6298, 0), v100, z5, tool0;
MoveL Offs(p0,174.0,105.2, 0), v100, z5, tool0;
MoveL Offs(p0,174.0,105.2, 0), v100, z5, tool0;
MoveJ Offs(p0,77.6,94.3, 10), v100, z1, tool0;
MoveL Offs(p0,78.40990000000002,93.33400000000002, 0), v100, z5, tool0;
MoveL Offs(p0,79.03920000000002,92.52400000000002, 0), v100, z5, tool0;
MoveL Offs(p0,79.4873,91.852, 0), v100, z5, tool0;
MoveL Offs(p0,79.7536,91.3, 0), v100, z5, tool0;
MoveL Offs(p0,79.8375,90.85, 0), v100, z5, tool0;
MoveL Offs(p0,79.7384,90.484, 0), v100, z5, tool0;
MoveL Offs(p0,79.45570000000001,90.184, 0), v100, z5, tool0;
MoveL Offs(p0,78.9888,89.932, 0), v100, z5, tool0;
MoveL Offs(p0,78.33709999999999,89.71000000000001, 0), v100, z5, tool0;
MoveL Offs(p0,76.0672,89.2084, 0), v100, z5, tool0;
MoveL Offs(p0,75.5384,89.1048, 0), v100, z5, tool0;
MoveL Offs(p0,75.0,89.0, 0), v100, z5, tool0;
MoveL Offs(p0,74.4616,88.8952, 0), v100, z5, tool0;
MoveL Offs(p0,73.9328,88.79159999999999, 0), v100, z5, tool0;
MoveL Offs(p0,73.42320000000001,88.69040000000001, 0), v100, z5, tool0;
MoveL Offs(p0,72.94239999999999,88.5928, 0), v100, z5, tool0;
MoveL Offs(p0,72.5,88.5, 0), v100, z5, tool0;
MoveL Offs(p0,71.01520000000001,88.284, 0), v100, z5, tool0;
MoveL Offs(p0,70.725,88.275, 0), v100, z5, tool0;
MoveL Offs(p0,70.4768,88.28399999999999, 0), v100, z5, tool0;
MoveL Offs(p0,70.34880000000001,89.59600000000003, 0), v100, z5, tool0;
MoveL Offs(p0,70.7317,90.273, 0), v100, z5, tool0;
MoveL Offs(p0,71.2064,90.98, 0), v100, z5, tool0;
MoveL Offs(p0,71.7375,91.675, 0), v100, z5, tool0;
MoveL Offs(p0,72.2896,92.31599999999999, 0), v100, z5, tool0;
MoveL Offs(p0,72.8273,92.86099999999999, 0), v100, z5, tool0;
MoveL Offs(p0,73.3152,93.268, 0), v100, z5, tool0;
MoveL Offs(p0,73.7179,93.495, 0), v100, z5, tool0;
MoveL Offs(p0,74.0,93.5, 0), v100, z5, tool0;
MoveL Offs(p0,74.45,93.725, 0), v100, z5, tool0;
MoveL Offs(p0,74.46799999999999,93.91040000000001, 0), v100, z5, tool0;
MoveL Offs(p0,74.462,94.13419999999999, 0), v100, z5, tool0;
MoveL Offs(p0,74.43200000000002,94.39280000000001, 0), v100, z5, tool0;
MoveL Offs(p0,74.378,94.68260000000001, 0), v100, z5, tool0;
MoveL Offs(p0,74.3,95.0, 0), v100, z5, tool0;
MoveL Offs(p0,74.6375,96.9, 0), v100, z5, tool0;
MoveL Offs(p0,75.02720000000001,96.73519999999999, 0), v100, z5, tool0;
MoveL Offs(p0,75.5201,96.3916, 0), v100, z5, tool0;
MoveL Offs(p0,76.1144,95.8704, 0), v100, z5, tool0;
MoveL Offs(p0,77.6,94.3, 0), v100, z5, tool0;
MoveL Offs(p0,77.6,94.3, 0), v100, z5, tool0;
MoveJ Offs(p0,153.0,86.0, 10), v100, z1, tool0;
MoveL Offs(p0,152.7057,82.27399999999999, 0), v100, z5, tool0;
MoveL Offs(p0,152.4144,81.47200000000001, 0), v100, z5, tool0;
MoveL Offs(p0,151.9875,80.85, 0), v100, z5, tool0;
MoveL Offs(p0,151.4016,80.38399999999999, 0), v100, z5, tool0;
MoveL Offs(p0,150.63330000000002,80.05, 0), v100, z5, tool0;
MoveL Offs(p0,149.6592,79.824, 0), v100, z5, tool0;
MoveL Offs(p0,148.45589999999999,79.682, 0), v100, z5, tool0;
MoveL Offs(p0,147.0,79.6, 0), v100, z5, tool0;
MoveL Offs(p0,145.45600000000002,79.3904, 0), v100, z5, tool0;
MoveL Offs(p0,145.175,79.3125, 0), v100, z5, tool0;
MoveL Offs(p0,144.948,79.22560000000001, 0), v100, z5, tool0;
MoveL Offs(p0,144.781,79.13029999999999, 0), v100, z5, tool0;
MoveL Offs(p0,144.68,79.0272, 0), v100, z5, tool0;
MoveL Offs(p0,144.651,78.91690000000001, 0), v100, z5, tool0;
MoveL Offs(p0,144.7,78.8, 0), v100, z5, tool0;
MoveL Offs(p0,144.3736,78.0528, 0), v100, z5, tool0;
MoveL Offs(p0,144.1375,77.8375, 0), v100, z5, tool0;
MoveL Offs(p0,143.8504,77.6192, 0), v100, z5, tool0;
MoveL Offs(p0,143.5177,77.40209999999999, 0), v100, z5, tool0;
MoveL Offs(p0,143.1448,77.19040000000001, 0), v100, z5, tool0;
MoveL Offs(p0,142.7371,76.98830000000001, 0), v100, z5, tool0;
MoveL Offs(p0,142.3,76.8, 0), v100, z5, tool0;
MoveL Offs(p0,140.6039,75.944, 0), v100, z5, tool0;
MoveL Offs(p0,138.89520000000002,74.89600000000003, 0), v100, z5, tool0;
MoveL Offs(p0,137.2033,73.686, 0), v100, z5, tool0;
MoveL Offs(p0,135.5576,72.34400000000001, 0), v100, z5, tool0;
MoveL Offs(p0,133.9875,70.9, 0), v100, z5, tool0;
MoveL Offs(p0,132.5224,69.384, 0), v100, z5, tool0;
MoveL Offs(p0,131.1917,67.826, 0), v100, z5, tool0;
MoveL Offs(p0,130.0248,66.256, 0), v100, z5, tool0;
MoveL Offs(p0,129.0511,64.704, 0), v100, z5, tool0;
MoveL Offs(p0,128.3,63.2, 0), v100, z5, tool0;
MoveL Offs(p0,127.95200000000003,62.3442, 0), v100, z5, tool0;
MoveL Offs(p0,127.68800000000006,61.621600000000015, 0), v100, z5, tool0;
MoveL Offs(p0,127.508,61.00940000000001, 0), v100, z5, tool0;
MoveL Offs(p0,127.412,60.48480000000001, 0), v100, z5, tool0;
MoveL Offs(p0,127.4,60.025, 0), v100, z5, tool0;
MoveL Offs(p0,127.47200000000001,59.6072, 0), v100, z5, tool0;
MoveL Offs(p0,127.628,59.208600000000004, 0), v100, z5, tool0;
MoveL Offs(p0,127.86800000000001,58.80640000000001, 0), v100, z5, tool0;
MoveL Offs(p0,128.6,57.9, 0), v100, z5, tool0;
MoveL Offs(p0,128.9335,57.592000000000006, 0), v100, z5, tool0;
MoveL Offs(p0,129.38400000000004,57.27200000000001, 0), v100, z5, tool0;
MoveL Offs(p0,129.9365,56.946000000000005, 0), v100, z5, tool0;
MoveL Offs(p0,130.576,56.620000000000005, 0), v100, z5, tool0;
MoveL Offs(p0,131.2875,56.3, 0), v100, z5, tool0;
MoveL Offs(p0,132.056,55.992, 0), v100, z5, tool0;
MoveL Offs(p0,132.8665,55.702, 0), v100, z5, tool0;
MoveL Offs(p0,133.704,55.436000000000014, 0), v100, z5, tool0;
MoveL Offs(p0,134.5535,55.2, 0), v100, z5, tool0;
MoveL Offs(p0,135.4,55.0, 0), v100, z5, tool0;
MoveL Offs(p0,136.81040000000002,54.734300000000005, 0), v100, z5, tool0;
MoveL Offs(p0,138.11520000000007,54.54240000000002, 0), v100, z5, tool0;
MoveL Offs(p0,139.42479999999998,54.432100000000005, 0), v100, z5, tool0;
MoveL Offs(p0,140.8496,54.41120000000001, 0), v100, z5, tool0;
MoveL Offs(p0,142.5,54.4875, 0), v100, z5, tool0;
MoveL Offs(p0,144.4864,54.6688, 0), v100, z5, tool0;
MoveL Offs(p0,149.9088,55.37760000000001, 0), v100, z5, tool0;
MoveL Offs(p0,153.56560000000002,55.9207, 0), v100, z5, tool0;
MoveL Offs(p0,158.0,56.6, 0), v100, z5, tool0;
MoveL Offs(p0,159.64080000000004,56.83760000000002, 0), v100, z5, tool0;
MoveL Offs(p0,160.2887,56.848400000000005, 0), v100, z5, tool0;
MoveL Offs(p0,161.8376,56.3192, 0), v100, z5, tool0;
MoveL Offs(p0,162.3043,55.9196, 0), v100, z5, tool0;
MoveL Offs(p0,162.78720000000004,55.3904, 0), v100, z5, tool0;
MoveL Offs(p0,163.3109,54.7208, 0), v100, z5, tool0;
MoveL Offs(p0,163.9,53.9, 0), v100, z5, tool0;
MoveL Offs(p0,164.32710000000003,53.30800000000001, 0), v100, z5, tool0;
MoveL Offs(p0,164.82080000000005,52.68000000000001, 0), v100, z5, tool0;
MoveL Offs(p0,165.3697,52.028, 0), v100, z5, tool0;
MoveL Offs(p0,165.96240000000003,51.364, 0), v100, z5, tool0;
MoveL Offs(p0,166.5875,50.7, 0), v100, z5, tool0;
MoveL Offs(p0,167.2336,50.048, 0), v100, z5, tool0;
MoveL Offs(p0,167.8893,49.42, 0), v100, z5, tool0;
MoveL Offs(p0,168.5432,48.828, 0), v100, z5, tool0;
MoveL Offs(p0,169.1839,48.284000000000006, 0), v100, z5, tool0;
MoveL Offs(p0,169.8,47.8, 0), v100, z5, tool0;
MoveL Offs(p0,173.3,45.0, 0), v100, z5, tool0;
MoveL Offs(p0,167.4,45.0, 0), v100, z5, tool0;
MoveL Offs(p0,163.0768,44.7856, 0), v100, z5, tool0;
MoveL Offs(p0,161.9375,44.675, 0), v100, z5, tool0;
MoveL Offs(p0,160.81919999999997,44.546400000000006, 0), v100, z5, tool0;
MoveL Offs(p0,159.74409999999997,44.40219999999999, 0), v100, z5, tool0;
MoveL Offs(p0,158.7344,44.244800000000005, 0), v100, z5, tool0;
MoveL Offs(p0,157.8123,44.076600000000006, 0), v100, z5, tool0;
MoveL Offs(p0,157.0,43.9, 0), v100, z5, tool0;
MoveL Offs(p0,156.2461,43.696200000000005, 0), v100, z5, tool0;
MoveL Offs(p0,155.49280000000005,43.505600000000015, 0), v100, z5, tool0;
MoveL Offs(p0,154.7527,43.3294, 0), v100, z5, tool0;
MoveL Offs(p0,154.0384,43.1688, 0), v100, z5, tool0;
MoveL Offs(p0,153.3625,43.025, 0), v100, z5, tool0;
MoveL Offs(p0,152.7376,42.89919999999999, 0), v100, z5, tool0;
MoveL Offs(p0,152.1763,42.79259999999999, 0), v100, z5, tool0;
MoveL Offs(p0,151.69120000000004,42.7064, 0), v100, z5, tool0;
MoveL Offs(p0,151.2949,42.6418, 0), v100, z5, tool0;
MoveL Offs(p0,151.0,42.6, 0), v100, z5, tool0;
MoveL Offs(p0,149.5258,42.254000000000005, 0), v100, z5, tool0;
MoveL Offs(p0,147.7384,41.60800000000001, 0), v100, z5, tool0;
MoveL Offs(p0,145.7206,40.709999999999994, 0), v100, z5, tool0;
MoveL Offs(p0,143.5552,39.608000000000004, 0), v100, z5, tool0;
MoveL Offs(p0,141.325,38.35, 0), v100, z5, tool0;
MoveL Offs(p0,139.11280000000002,36.984, 0), v100, z5, tool0;
MoveL Offs(p0,137.0014,35.55800000000001, 0), v100, z5, tool0;
MoveL Offs(p0,135.0736,34.120000000000005, 0), v100, z5, tool0;
MoveL Offs(p0,133.4122,32.718, 0), v100, z5, tool0;
MoveL Offs(p0,132.1,31.4, 0), v100, z5, tool0;
MoveL Offs(p0,128.1,26.9, 0), v100, z5, tool0;
MoveL Offs(p0,126.0,31.7, 0), v100, z5, tool0;
MoveL Offs(p0,125.62920000000001,32.533300000000004, 0), v100, z5, tool0;
MoveL Offs(p0,125.24160000000002,33.458400000000005, 0), v100, z5, tool0;
MoveL Offs(p0,124.8444,34.45309999999999, 0), v100, z5, tool0;
MoveL Offs(p0,124.44480000000001,35.495200000000004, 0), v100, z5, tool0;
MoveL Offs(p0,124.05,36.5625, 0), v100, z5, tool0;
MoveL Offs(p0,123.66720000000001,37.632799999999996, 0), v100, z5, tool0;
MoveL Offs(p0,123.3036,38.6839, 0), v100, z5, tool0;
MoveL Offs(p0,122.96640000000002,39.6936, 0), v100, z5, tool0;
MoveL Offs(p0,122.66280000000002,40.639700000000005, 0), v100, z5, tool0;
MoveL Offs(p0,122.4,41.5, 0), v100, z5, tool0;
MoveL Offs(p0,121.95950000000002,43.493700000000004, 0), v100, z5, tool0;
MoveL Offs(p0,121.60000000000002,45.893600000000006, 0), v100, z5, tool0;
MoveL Offs(p0,121.32449999999999,48.547900000000006, 0), v100, z5, tool0;
MoveL Offs(p0,121.136,51.3048, 0), v100, z5, tool0;
MoveL Offs(p0,121.0375,54.0125, 0), v100, z5, tool0;
MoveL Offs(p0,121.032,56.5192, 0), v100, z5, tool0;
MoveL Offs(p0,121.12249999999999,58.6731, 0), v100, z5, tool0;
MoveL Offs(p0,121.31200000000001,60.3224, 0), v100, z5, tool0;
MoveL Offs(p0,121.60350000000001,61.3153, 0), v100, z5, tool0;
MoveL Offs(p0,122.0,61.5, 0), v100, z5, tool0;
MoveL Offs(p0,122.5404,61.7177, 0), v100, z5, tool0;
MoveL Offs(p0,122.52159999999999,61.8808, 0), v100, z5, tool0;
MoveL Offs(p0,122.4752,62.0751, 0), v100, z5, tool0;
MoveL Offs(p0,122.4,62.3, 0), v100, z5, tool0;
MoveL Offs(p0,123.05969999999999,65.8856, 0), v100, z5, tool0;
MoveL Offs(p0,123.78240000000001,67.6232, 0), v100, z5, tool0;
MoveL Offs(p0,124.6875,69.5, 0), v100, z5, tool0;
MoveL Offs(p0,125.7336,71.43679999999999, 0), v100, z5, tool0;
MoveL Offs(p0,126.87930000000001,73.35440000000001, 0), v100, z5, tool0;
MoveL Offs(p0,128.0832,75.17360000000001, 0), v100, z5, tool0;
MoveL Offs(p0,129.30390000000003,76.8152, 0), v100, z5, tool0;
MoveL Offs(p0,130.5,78.2, 0), v100, z5, tool0;
MoveL Offs(p0,132.1072,79.74740000000001, 0), v100, z5, tool0;
MoveL Offs(p0,133.88960000000003,81.30320000000002, 0), v100, z5, tool0;
MoveL Offs(p0,135.78839999999997,82.8278, 0), v100, z5, tool0;
MoveL Offs(p0,137.7448,84.2816, 0), v100, z5, tool0;
MoveL Offs(p0,139.7,85.625, 0), v100, z5, tool0;
MoveL Offs(p0,141.5952,86.8184, 0), v100, z5, tool0;
MoveL Offs(p0,143.3716,87.8222, 0), v100, z5, tool0;
MoveL Offs(p0,144.9704,88.5968, 0), v100, z5, tool0;
MoveL Offs(p0,146.3328,89.10260000000001, 0), v100, z5, tool0;
MoveL Offs(p0,147.4,89.3, 0), v100, z5, tool0;
MoveL Offs(p0,148.92000000000002,89.55120000000001, 0), v100, z5, tool0;
MoveL Offs(p0,149.225,89.65, 0), v100, z5, tool0;
MoveL Offs(p0,149.488,89.7608, 0), v100, z5, tool0;
MoveL Offs(p0,149.703,89.8824, 0), v100, z5, tool0;
MoveL Offs(p0,149.864,90.01360000000001, 0), v100, z5, tool0;
MoveL Offs(p0,149.965,90.1532, 0), v100, z5, tool0;
MoveL Offs(p0,150.0,90.3, 0), v100, z5, tool0;
MoveL Offs(p0,150.29760000000002,90.71920000000001, 0), v100, z5, tool0;
MoveL Offs(p0,150.45,90.8, 0), v100, z5, tool0;
MoveL Offs(p0,150.62640000000002,90.8688, 0), v100, z5, tool0;
MoveL Offs(p0,150.82319999999999,90.92439999999999, 0), v100, z5, tool0;
MoveL Offs(p0,151.0368,90.96560000000001, 0), v100, z5, tool0;
MoveL Offs(p0,151.26360000000003,90.9912, 0), v100, z5, tool0;
MoveL Offs(p0,151.5,91.0, 0), v100, z5, tool0;
MoveL Offs(p0,152.3091,90.63820000000001, 0), v100, z5, tool0;
MoveL Offs(p0,152.50320000000002,90.3344, 0), v100, z5, tool0;
MoveL Offs(p0,152.6625,89.925, 0), v100, z5, tool0;
MoveL Offs(p0,152.7888,89.4016, 0), v100, z5, tool0;
MoveL Offs(p0,152.88389999999998,88.7558, 0), v100, z5, tool0;
MoveL Offs(p0,152.9496,87.97920000000002, 0), v100, z5, tool0;
MoveL Offs(p0,152.9877,87.0634, 0), v100, z5, tool0;
MoveL Offs(p0,153.0,86.0, 0), v100, z5, tool0;
MoveL Offs(p0,153.0,86.0, 0), v100, z5, tool0;
MoveJ Offs(p0,256.0,84.5, 10), v100, z1, tool0;
MoveL Offs(p0,255.7520000000001,81.46560000000002, 0), v100, z5, tool0;
MoveL Offs(p0,255.46000000000004,79.67689999999999, 0), v100, z5, tool0;
MoveL Offs(p0,255.07200000000003,77.7688, 0), v100, z5, tool0;
MoveL Offs(p0,254.6,75.7875, 0), v100, z5, tool0;
MoveL Offs(p0,254.05599999999998,73.7792, 0), v100, z5, tool0;
MoveL Offs(p0,253.452,71.79010000000001, 0), v100, z5, tool0;
MoveL Offs(p0,252.8,69.8664, 0), v100, z5, tool0;
MoveL Offs(p0,252.112,68.0543, 0), v100, z5, tool0;
MoveL Offs(p0,251.4,66.4, 0), v100, z5, tool0;
MoveL Offs(p0,249.63530000000006,63.032900000000005, 0), v100, z5, tool0;
MoveL Offs(p0,247.5904000000001,59.839200000000005, 0), v100, z5, tool0;
MoveL Offs(p0,245.27909999999997,56.8303, 0), v100, z5, tool0;
MoveL Offs(p0,242.7152,54.0176, 0), v100, z5, tool0;
MoveL Offs(p0,239.9125,51.4125, 0), v100, z5, tool0;
MoveL Offs(p0,236.88479999999998,49.0264, 0), v100, z5, tool0;
MoveL Offs(p0,233.64589999999998,46.87069999999999, 0), v100, z5, tool0;
MoveL Offs(p0,230.20960000000005,44.9568, 0), v100, z5, tool0;
MoveL Offs(p0,226.5897,43.2961, 0), v100, z5, tool0;
MoveL Offs(p0,222.8,41.9, 0), v100, z5, tool0;
MoveL Offs(p0,218.31120000000004,40.7153, 0), v100, z5, tool0;
MoveL Offs(p0,213.37360000000007,39.91040000000001, 0), v100, z5, tool0;
MoveL Offs(p0,208.18039999999996,39.4691, 0), v100, z5, tool0;
MoveL Offs(p0,202.92480000000003,39.3752, 0), v100, z5, tool0;
MoveL Offs(p0,197.8,39.6125, 0), v100, z5, tool0;
MoveL Offs(p0,192.99919999999997,40.1648, 0), v100, z5, tool0;
MoveL Offs(p0,188.7156,41.0159, 0), v100, z5, tool0;
MoveL Offs(p0,185.1424,42.14960000000001, 0), v100, z5, tool0;
MoveL Offs(p0,182.4728,43.5497, 0), v100, z5, tool0;
MoveL Offs(p0,180.9,45.2, 0), v100, z5, tool0;
MoveL Offs(p0,180.47950000000003,46.2793, 0), v100, z5, tool0;
MoveL Offs(p0,180.17600000000004,47.67840000000001, 0), v100, z5, tool0;
MoveL Offs(p0,179.98649999999998,49.339099999999995, 0), v100, z5, tool0;
MoveL Offs(p0,179.90800000000002,51.2032, 0), v100, z5, tool0;
MoveL Offs(p0,179.9375,53.2125, 0), v100, z5, tool0;
MoveL Offs(p0,180.07200000000003,55.308800000000005, 0), v100, z5, tool0;
MoveL Offs(p0,180.30849999999998,57.433899999999994, 0), v100, z5, tool0;
MoveL Offs(p0,180.644,59.5296, 0), v100, z5, tool0;
MoveL Offs(p0,181.6,63.4, 0), v100, z5, tool0;
MoveL Offs(p0,182.45130000000003,65.4424, 0), v100, z5, tool0;
MoveL Offs(p0,183.64640000000003,67.57120000000002, 0), v100, z5, tool0;
MoveL Offs(p0,185.12709999999998,69.7288, 0), v100, z5, tool0;
MoveL Offs(p0,186.83520000000001,71.8576, 0), v100, z5, tool0;
MoveL Offs(p0,188.7125,73.9, 0), v100, z5, tool0;
MoveL Offs(p0,190.7008,75.79839999999999, 0), v100, z5, tool0;
MoveL Offs(p0,192.7419,77.4952, 0), v100, z5, tool0;
MoveL Offs(p0,194.7776,78.93280000000001, 0), v100, z5, tool0;
MoveL Offs(p0,196.7497,80.0536, 0), v100, z5, tool0;
MoveL Offs(p0,198.6,80.8, 0), v100, z5, tool0;
MoveL Offs(p0,199.6073,81.0669, 0), v100, z5, tool0;
MoveL Offs(p0,200.55040000000005,81.26720000000003, 0), v100, z5, tool0;
MoveL Offs(p0,201.4611,81.40029999999999, 0), v100, z5, tool0;
MoveL Offs(p0,202.37120000000002,81.46560000000001, 0), v100, z5, tool0;
MoveL Offs(p0,203.3125,81.4625, 0), v100, z5, tool0;
MoveL Offs(p0,204.3168,81.39040000000001, 0), v100, z5, tool0;
MoveL Offs(p0,205.41590000000002,81.2487, 0), v100, z5, tool0;
MoveL Offs(p0,206.6416,81.0368, 0), v100, z5, tool0;
MoveL Offs(p0,209.6,80.4, 0), v100, z5, tool0;
MoveL Offs(p0,214.0483,79.53780000000002, 0), v100, z5, tool0;
MoveL Offs(p0,218.64240000000004,78.98640000000003, 0), v100, z5, tool0;
MoveL Offs(p0,223.30610000000001,78.73859999999999, 0), v100, z5, tool0;
MoveL Offs(p0,227.9632,78.78720000000001, 0), v100, z5, tool0;
MoveL Offs(p0,232.5375,79.125, 0), v100, z5, tool0;
MoveL Offs(p0,236.95279999999997,79.7448, 0), v100, z5, tool0;
MoveL Offs(p0,241.1329,80.6394, 0), v100, z5, tool0;
MoveL Offs(p0,245.00160000000005,81.80160000000001, 0), v100, z5, tool0;
MoveL Offs(p0,248.48270000000002,83.2242, 0), v100, z5, tool0;
MoveL Offs(p0,251.5,84.9, 0), v100, z5, tool0;
MoveL Offs(p0,252.598,85.5989, 0), v100, z5, tool0;
MoveL Offs(p0,253.50400000000008,86.13520000000003, 0), v100, z5, tool0;
MoveL Offs(p0,254.23599999999996,86.50829999999999, 0), v100, z5, tool0;
MoveL Offs(p0,254.81200000000004,86.7176, 0), v100, z5, tool0;
MoveL Offs(p0,255.25,86.7625, 0), v100, z5, tool0;
MoveL Offs(p0,255.56800000000004,86.6424, 0), v100, z5, tool0;
MoveL Offs(p0,255.78400000000002,86.3567, 0), v100, z5, tool0;
MoveL Offs(p0,255.916,85.9048, 0), v100, z5, tool0;
MoveL Offs(p0,255.98200000000003,85.2861, 0), v100, z5, tool0;
MoveL Offs(p0,256.0,84.5, 0), v100, z5, tool0;
MoveL Offs(p0,256.0,84.5, 0), v100, z5, tool0;
MoveJ Offs(p0,92.7,84.8, 10), v100, z1, tool0;
MoveL Offs(p0,93.62400000000004,84.44400000000002, 0), v100, z5, tool0;
MoveL Offs(p0,94.09049999999999,84.27349999999998, 0), v100, z5, tool0;
MoveL Offs(p0,94.548,84.11200000000001, 0), v100, z5, tool0;
MoveL Offs(p0,94.9875,83.9625, 0), v100, z5, tool0;
MoveL Offs(p0,95.39999999999999,83.828, 0), v100, z5, tool0;
MoveL Offs(p0,95.7765,83.7115, 0), v100, z5, tool0;
MoveL Offs(p0,96.108,83.61600000000001, 0), v100, z5, tool0;
MoveL Offs(p0,96.38550000000001,83.5445, 0), v100, z5, tool0;
MoveL Offs(p0,96.6,83.5, 0), v100, z5, tool0;
MoveL Offs(p0,97.3992,83.1985, 0), v100, z5, tool0;
MoveL Offs(p0,97.75840000000001,83.052, 0), v100, z5, tool0;
MoveL Offs(p0,98.15,82.8875, 0), v100, z5, tool0;
MoveL Offs(p0,98.56559999999999,82.708, 0), v100, z5, tool0;
MoveL Offs(p0,98.9968,82.5165, 0), v100, z5, tool0;
MoveL Offs(p0,99.43520000000001,82.316, 0), v100, z5, tool0;
MoveL Offs(p0,99.87240000000001,82.1095, 0), v100, z5, tool0;
MoveL Offs(p0,100.3,81.9, 0), v100, z5, tool0;
MoveL Offs(p0,102.9,80.5, 0), v100, z5, tool0;
MoveL Offs(p0,97.5,77.6, 0), v100, z5, tool0;
MoveL Offs(p0,95.9544,76.7415, 0), v100, z5, tool0;
MoveL Offs(p0,94.38720000000004,75.73600000000002, 0), v100, z5, tool0;
MoveL Offs(p0,92.8128,74.5985, 0), v100, z5, tool0;
MoveL Offs(p0,91.2456,73.34400000000001, 0), v100, z5, tool0;
MoveL Offs(p0,89.7,71.9875, 0), v100, z5, tool0;
MoveL Offs(p0,88.19039999999998,70.54400000000001, 0), v100, z5, tool0;
MoveL Offs(p0,86.73119999999999,69.0285, 0), v100, z5, tool0;
MoveL Offs(p0,85.33680000000001,67.456, 0), v100, z5, tool0;
MoveL Offs(p0,84.0216,65.84150000000001, 0), v100, z5, tool0;
MoveL Offs(p0,82.8,64.2, 0), v100, z5, tool0;
MoveL Offs(p0,82.40480000000001,63.65340000000001, 0), v100, z5, tool0;
MoveL Offs(p0,82.05040000000001,63.211200000000005, 0), v100, z5, tool0;
MoveL Offs(p0,81.72359999999999,62.8698, 0), v100, z5, tool0;
MoveL Offs(p0,81.41120000000001,62.625600000000006, 0), v100, z5, tool0;
MoveL Offs(p0,81.1,62.475, 0), v100, z5, tool0;
MoveL Offs(p0,80.77680000000001,62.414399999999986, 0), v100, z5, tool0;
MoveL Offs(p0,80.42840000000001,62.440200000000004, 0), v100, z5, tool0;
MoveL Offs(p0,80.0416,62.54880000000001, 0), v100, z5, tool0;
MoveL Offs(p0,79.6032,62.736599999999996, 0), v100, z5, tool0;
MoveL Offs(p0,79.1,63.0, 0), v100, z5, tool0;
MoveL Offs(p0,77.94280000000002,63.46900000000001, 0), v100, z5, tool0;
MoveL Offs(p0,76.34640000000002,63.908000000000015, 0), v100, z5, tool0;
MoveL Offs(p0,74.4236,64.305, 0), v100, z5, tool0;
MoveL Offs(p0,72.28720000000001,64.64800000000001, 0), v100, z5, tool0;
MoveL Offs(p0,70.05,64.925, 0), v100, z5, tool0;
MoveL Offs(p0,67.82480000000001,65.124, 0), v100, z5, tool0;
MoveL Offs(p0,65.72439999999999,65.233, 0), v100, z5, tool0;
MoveL Offs(p0,63.861599999999996,65.24000000000001, 0), v100, z5, tool0;
MoveL Offs(p0,62.34920000000001,65.133, 0), v100, z5, tool0;
MoveL Offs(p0,61.3,64.9, 0), v100, z5, tool0;
MoveL Offs(p0,60.21250000000001,64.2844, 0), v100, z5, tool0;
MoveL Offs(p0,59.46400000000001,63.41920000000001, 0), v100, z5, tool0;
MoveL Offs(p0,59.04549999999999,62.336800000000004, 0), v100, z5, tool0;
MoveL Offs(p0,58.948000000000015,61.069599999999994, 0), v100, z5, tool0;
MoveL Offs(p0,59.1625,59.65, 0), v100, z5, tool0;
MoveL Offs(p0,59.67999999999999,58.110400000000006, 0), v100, z5, tool0;
MoveL Offs(p0,60.49150000000001,56.4832, 0), v100, z5, tool0;
MoveL Offs(p0,61.58800000000001,54.8008, 0), v100, z5, tool0;
MoveL Offs(p0,62.9605,53.095600000000005, 0), v100, z5, tool0;
MoveL Offs(p0,64.6,51.4, 0), v100, z5, tool0;
MoveL Offs(p0,64.97150000000002,51.03800000000001, 0), v100, z5, tool0;
MoveL Offs(p0,65.30400000000002,50.676000000000016, 0), v100, z5, tool0;
MoveL Offs(p0,65.59450000000001,50.32000000000001, 0), v100, z5, tool0;
MoveL Offs(p0,65.84,49.976000000000006, 0), v100, z5, tool0;
MoveL Offs(p0,66.0375,49.65, 0), v100, z5, tool0;
MoveL Offs(p0,66.184,49.348, 0), v100, z5, tool0;
MoveL Offs(p0,66.2765,49.076, 0), v100, z5, tool0;
MoveL Offs(p0,66.31200000000001,48.84, 0), v100, z5, tool0;
MoveL Offs(p0,66.2875,48.646, 0), v100, z5, tool0;
MoveL Offs(p0,66.2,48.5, 0), v100, z5, tool0;
MoveL Offs(p0,65.9939,48.218300000000006, 0), v100, z5, tool0;
MoveL Offs(p0,65.98880000000001,48.1576, 0), v100, z5, tool0;
MoveL Offs(p0,66.5,48.1, 0), v100, z5, tool0;
MoveL Offs(p0,67.9272,47.821600000000004, 0), v100, z5, tool0;
MoveL Offs(p0,68.4625,47.6125, 0), v100, z5, tool0;
MoveL Offs(p0,69.0488,47.3584, 0), v100, z5, tool0;
MoveL Offs(p0,69.6759,47.0647, 0), v100, z5, tool0;
MoveL Offs(p0,70.3336,46.7368, 0), v100, z5, tool0;
MoveL Offs(p0,71.0117,46.380100000000006, 0), v100, z5, tool0;
MoveL Offs(p0,71.7,46.0, 0), v100, z5, tool0;
MoveL Offs(p0,72.7681,45.356300000000005, 0), v100, z5, tool0;
MoveL Offs(p0,73.64480000000002,44.786400000000015, 0), v100, z5, tool0;
MoveL Offs(p0,74.3487,44.2621, 0), v100, z5, tool0;
MoveL Offs(p0,74.89840000000001,43.75520000000001, 0), v100, z5, tool0;
MoveL Offs(p0,75.3125,43.2375, 0), v100, z5, tool0;
MoveL Offs(p0,75.6096,42.6808, 0), v100, z5, tool0;
MoveL Offs(p0,75.8083,42.0569, 0), v100, z5, tool0;
MoveL Offs(p0,75.92720000000001,41.337599999999995, 0), v100, z5, tool0;
MoveL Offs(p0,75.98490000000001,40.4947, 0), v100, z5, tool0;
MoveL Offs(p0,76.0,39.5, 0), v100, z5, tool0;
MoveL Offs(p0,76.2625,35.7, 0), v100, z5, tool0;
MoveL Offs(p0,76.3672,34.913599999999995, 0), v100, z5, tool0;
MoveL Offs(p0,76.48509999999999,34.1548, 0), v100, z5, tool0;
MoveL Offs(p0,76.6144,33.43920000000001, 0), v100, z5, tool0;
MoveL Offs(p0,76.75330000000001,32.7824, 0), v100, z5, tool0;
MoveL Offs(p0,76.9,32.2, 0), v100, z5, tool0;
MoveL Offs(p0,77.16320000000002,31.214400000000005, 0), v100, z5, tool0;
MoveL Offs(p0,77.26629999999999,30.759099999999997, 0), v100, z5, tool0;
MoveL Offs(p0,77.34960000000001,30.339199999999998, 0), v100, z5, tool0;
MoveL Offs(p0,77.4125,29.9625, 0), v100, z5, tool0;
MoveL Offs(p0,77.45439999999999,29.6368, 0), v100, z5, tool0;
MoveL Offs(p0,77.47470000000001,29.3699, 0), v100, z5, tool0;
MoveL Offs(p0,77.4728,29.169600000000003, 0), v100, z5, tool0;
MoveL Offs(p0,77.4481,29.0437, 0), v100, z5, tool0;
MoveL Offs(p0,77.4,29.0, 0), v100, z5, tool0;
MoveL Offs(p0,76.12640000000002,29.473600000000012, 0), v100, z5, tool0;
MoveL Offs(p0,75.0726,29.990899999999993, 0), v100, z5, tool0;
MoveL Offs(p0,73.8592,30.628800000000002, 0), v100, z5, tool0;
MoveL Offs(p0,72.575,31.3375, 0), v100, z5, tool0;
MoveL Offs(p0,71.30879999999999,32.0672, 0), v100, z5, tool0;
MoveL Offs(p0,70.14939999999999,32.768100000000004, 0), v100, z5, tool0;
MoveL Offs(p0,69.1856,33.39040000000001, 0), v100, z5, tool0;
MoveL Offs(p0,68.5062,33.8843, 0), v100, z5, tool0;
MoveL Offs(p0,68.2,34.2, 0), v100, z5, tool0;
MoveL Offs(p0,67.8742,34.4547, 0), v100, z5, tool0;
MoveL Offs(p0,67.7104,34.4944, 0), v100, z5, tool0;
MoveL Offs(p0,67.525,34.5125, 0), v100, z5, tool0;
MoveL Offs(p0,67.3216,34.5096, 0), v100, z5, tool0;
MoveL Offs(p0,67.1038,34.48630000000001, 0), v100, z5, tool0;
MoveL Offs(p0,66.8752,34.443200000000004, 0), v100, z5, tool0;
MoveL Offs(p0,65.0176,34.6321, 0), v100, z5, tool0;
MoveL Offs(p0,65.0,34.8, 0), v100, z5, tool0;
MoveL Offs(p0,64.39120000000001,35.17280000000002, 0), v100, z5, tool0;
MoveL Offs(p0,63.687799999999996,35.279700000000005, 0), v100, z5, tool0;
MoveL Offs(p0,62.76959999999999,35.3344, 0), v100, z5, tool0;
MoveL Offs(p0,61.675,35.3375, 0), v100, z5, tool0;
MoveL Offs(p0,60.4424,35.2896, 0), v100, z5, tool0;
MoveL Offs(p0,59.1102,35.1913, 0), v100, z5, tool0;
MoveL Offs(p0,57.71680000000001,35.0432, 0), v100, z5, tool0;
MoveL Offs(p0,54.9,34.6, 0), v100, z5, tool0;
MoveL Offs(p0,53.26400000000001,35.34240000000001, 0), v100, z5, tool0;
MoveL Offs(p0,52.5015,36.4576, 0), v100, z5, tool0;
MoveL Offs(p0,51.79600000000001,37.995200000000004, 0), v100, z5, tool0;
MoveL Offs(p0,51.1625,39.9, 0), v100, z5, tool0;
MoveL Offs(p0,50.616,42.116800000000005, 0), v100, z5, tool0;
MoveL Offs(p0,50.171499999999995,44.5904, 0), v100, z5, tool0;
MoveL Offs(p0,49.84400000000001,47.265600000000006, 0), v100, z5, tool0;
MoveL Offs(p0,49.6485,50.08720000000001, 0), v100, z5, tool0;
MoveL Offs(p0,49.6,53.0, 0), v100, z5, tool0;
MoveL Offs(p0,49.99520000000002,58.940800000000024, 0), v100, z5, tool0;
MoveL Offs(p0,50.4568,61.6247, 0), v100, z5, tool0;
MoveL Offs(p0,51.10560000000001,64.1424, 0), v100, z5, tool0;
MoveL Offs(p0,51.95,66.5125, 0), v100, z5, tool0;
MoveL Offs(p0,52.998400000000004,68.7536, 0), v100, z5, tool0;
MoveL Offs(p0,54.2592,70.88430000000001, 0), v100, z5, tool0;
MoveL Offs(p0,55.740800000000014,72.92320000000002, 0), v100, z5, tool0;
MoveL Offs(p0,57.451600000000006,74.8889, 0), v100, z5, tool0;
MoveL Offs(p0,59.4,76.8, 0), v100, z5, tool0;
MoveL Offs(p0,61.5369,78.66140000000001, 0), v100, z5, tool0;
MoveL Offs(p0,63.64320000000002,80.29120000000003, 0), v100, z5, tool0;
MoveL Offs(p0,65.7423,81.69779999999999, 0), v100, z5, tool0;
MoveL Offs(p0,67.85760000000002,82.8896, 0), v100, z5, tool0;
MoveL Offs(p0,70.0125,83.875, 0), v100, z5, tool0;
MoveL Offs(p0,72.2304,84.66239999999999, 0), v100, z5, tool0;
MoveL Offs(p0,74.5347,85.26019999999998, 0), v100, z5, tool0;
MoveL Offs(p0,76.9488,85.6768, 0), v100, z5, tool0;
MoveL Offs(p0,79.4961,85.92060000000001, 0), v100, z5, tool0;
MoveL Offs(p0,82.2,86.0, 0), v100, z5, tool0;
MoveL Offs(p0,87.2496,85.7792, 0), v100, z5, tool0;
MoveL Offs(p0,88.425,85.6625, 0), v100, z5, tool0;
MoveL Offs(p0,89.5224,85.5248, 0), v100, z5, tool0;
MoveL Offs(p0,90.5202,85.3679, 0), v100, z5, tool0;
MoveL Offs(p0,91.39680000000001,85.1936, 0), v100, z5, tool0;
MoveL Offs(p0,92.1306,85.00370000000001, 0), v100, z5, tool0;
MoveL Offs(p0,92.7,84.8, 0), v100, z5, tool0;
MoveL Offs(p0,92.7,84.8, 0), v100, z5, tool0;
MoveJ Offs(p0,37.3,83.4, 10), v100, z1, tool0;
MoveL Offs(p0,37.894200000000005,83.05100000000002, 0), v100, z5, tool0;
MoveL Offs(p0,38.585600000000014,82.61200000000002, 0), v100, z5, tool0;
MoveL Offs(p0,39.3574,82.095, 0), v100, z5, tool0;
MoveL Offs(p0,40.192800000000005,81.512, 0), v100, z5, tool0;
MoveL Offs(p0,41.075,80.875, 0), v100, z5, tool0;
MoveL Offs(p0,41.9872,80.196, 0), v100, z5, tool0;
MoveL Offs(p0,42.9126,79.487, 0), v100, z5, tool0;
MoveL Offs(p0,43.8344,78.76, 0), v100, z5, tool0;
MoveL Offs(p0,44.7358,78.027, 0), v100, z5, tool0;
MoveL Offs(p0,45.6,77.3, 0), v100, z5, tool0;
MoveL Offs(p0,50.8,72.9, 0), v100, z5, tool0;
MoveL Offs(p0,48.9,68.0, 0), v100, z5, tool0;
MoveL Offs(p0,48.60380000000001,67.15330000000002, 0), v100, z5, tool0;
MoveL Offs(p0,48.31840000000001,66.3024, 0), v100, z5, tool0;
MoveL Offs(p0,48.04859999999999,65.4611, 0), v100, z5, tool0;
MoveL Offs(p0,47.7992,64.64320000000001, 0), v100, z5, tool0;
MoveL Offs(p0,47.575,63.8625, 0), v100, z5, tool0;
MoveL Offs(p0,47.3808,63.132799999999996, 0), v100, z5, tool0;
MoveL Offs(p0,47.2214,62.4679, 0), v100, z5, tool0;
MoveL Offs(p0,47.101600000000005,61.881600000000006, 0), v100, z5, tool0;
MoveL Offs(p0,47.0262,61.38770000000001, 0), v100, z5, tool0;
MoveL Offs(p0,47.0,61.0, 0), v100, z5, tool0;
MoveL Offs(p0,46.765,59.49950000000001, 0), v100, z5, tool0;
MoveL Offs(p0,46.10400000000001,58.74000000000001, 0), v100, z5, tool0;
MoveL Offs(p0,45.083,58.66450000000001, 0), v100, z5, tool0;
MoveL Offs(p0,43.76800000000001,59.215999999999994, 0), v100, z5, tool0;
MoveL Offs(p0,42.225,60.3375, 0), v100, z5, tool0;
MoveL Offs(p0,40.519999999999996,61.972, 0), v100, z5, tool0;
MoveL Offs(p0,38.718999999999994,64.0625, 0), v100, z5, tool0;
MoveL Offs(p0,36.888,66.552, 0), v100, z5, tool0;
MoveL Offs(p0,35.093,69.3835, 0), v100, z5, tool0;
MoveL Offs(p0,33.4,72.5, 0), v100, z5, tool0;
MoveL Offs(p0,32.57940000000001,74.17030000000001, 0), v100, z5, tool0;
MoveL Offs(p0,31.911200000000008,75.60240000000002, 0), v100, z5, tool0;
MoveL Offs(p0,31.3858,76.82809999999999, 0), v100, z5, tool0;
MoveL Offs(p0,30.993599999999997,77.87920000000001, 0), v100, z5, tool0;
MoveL Offs(p0,30.725,78.7875, 0), v100, z5, tool0;
MoveL Offs(p0,30.5704,79.5848, 0), v100, z5, tool0;
MoveL Offs(p0,30.5202,80.3029, 0), v100, z5, tool0;
MoveL Offs(p0,30.5648,80.9736, 0), v100, z5, tool0;
MoveL Offs(p0,30.6946,81.62870000000001, 0), v100, z5, tool0;
MoveL Offs(p0,30.9,82.3, 0), v100, z5, tool0;
MoveL Offs(p0,31.254700000000003,83.1435, 0), v100, z5, tool0;
MoveL Offs(p0,31.61360000000001,83.81600000000002, 0), v100, z5, tool0;
MoveL Offs(p0,31.998900000000003,84.3205, 0), v100, z5, tool0;
MoveL Offs(p0,32.4328,84.66, 0), v100, z5, tool0;
MoveL Offs(p0,32.9375,84.8375, 0), v100, z5, tool0;
MoveL Offs(p0,33.535199999999996,84.85600000000001, 0), v100, z5, tool0;
MoveL Offs(p0,34.2481,84.71849999999999, 0), v100, z5, tool0;
MoveL Offs(p0,35.098400000000005,84.428, 0), v100, z5, tool0;
MoveL Offs(p0,36.1083,83.98750000000001, 0), v100, z5, tool0;
MoveL Offs(p0,37.3,83.4, 0), v100, z5, tool0;
MoveL Offs(p0,37.3,83.4, 0), v100, z5, tool0;
MoveJ Offs(p0,124.7,78.6, 10), v100, z1, tool0;
MoveL Offs(p0,124.33040000000001,77.4976, 0), v100, z5, tool0;
MoveL Offs(p0,124.1,76.9625, 0), v100, z5, tool0;
MoveL Offs(p0,123.82159999999999,76.3464, 0), v100, z5, tool0;
MoveL Offs(p0,123.49879999999999,75.66069999999999, 0), v100, z5, tool0;
MoveL Offs(p0,123.13520000000001,74.91680000000001, 0), v100, z5, tool0;
MoveL Offs(p0,122.73440000000001,74.12610000000001, 0), v100, z5, tool0;
MoveL Offs(p0,122.3,73.3, 0), v100, z5, tool0;
MoveL Offs(p0,119.6,68.3, 0), v100, z5, tool0;
MoveL Offs(p0,113.1,67.6, 0), v100, z5, tool0;
MoveL Offs(p0,109.62780000000001,67.1075, 0), v100, z5, tool0;
MoveL Offs(p0,106.16640000000002,66.26400000000002, 0), v100, z5, tool0;
MoveL Offs(p0,102.7986,65.1205, 0), v100, z5, tool0;
MoveL Offs(p0,99.6072,63.72800000000001, 0), v100, z5, tool0;
MoveL Offs(p0,96.675,62.1375, 0), v100, z5, tool0;
MoveL Offs(p0,94.0848,60.4, 0), v100, z5, tool0;
MoveL Offs(p0,91.9194,58.5665, 0), v100, z5, tool0;
MoveL Offs(p0,90.26160000000002,56.68800000000001, 0), v100, z5, tool0;
MoveL Offs(p0,89.1942,54.8155, 0), v100, z5, tool0;
MoveL Offs(p0,88.8,53.0, 0), v100, z5, tool0;
MoveL Offs(p0,89.29680000000003,50.33680000000002, 0), v100, z5, tool0;
MoveL Offs(p0,90.0672,49.2317, 0), v100, z5, tool0;
MoveL Offs(p0,91.23840000000001,48.254400000000004, 0), v100, z5, tool0;
MoveL Offs(p0,92.85,47.3875, 0), v100, z5, tool0;
MoveL Offs(p0,94.94160000000001,46.6136, 0), v100, z5, tool0;
MoveL Offs(p0,97.5528,45.9153, 0), v100, z5, tool0;
MoveL Offs(p0,100.7232,45.275200000000005, 0), v100, z5, tool0;
MoveL Offs(p0,104.4924,44.6759, 0), v100, z5, tool0;
MoveL Offs(p0,108.9,44.1, 0), v100, z5, tool0;
MoveL Offs(p0,111.25200000000004,43.75760000000001, 0), v100, z5, tool0;
MoveL Offs(p0,112.36500000000001,43.560900000000004, 0), v100, z5, tool0;
MoveL Offs(p0,113.412,43.3528, 0), v100, z5, tool0;
MoveL Offs(p0,114.375,43.1375, 0), v100, z5, tool0;
MoveL Offs(p0,115.23600000000002,42.919200000000004, 0), v100, z5, tool0;
MoveL Offs(p0,115.977,42.702099999999994, 0), v100, z5, tool0;
MoveL Offs(p0,116.58000000000001,42.4904, 0), v100, z5, tool0;
MoveL Offs(p0,117.027,42.28830000000001, 0), v100, z5, tool0;
MoveL Offs(p0,117.3,42.1, 0), v100, z5, tool0;
MoveL Offs(p0,117.61010000000002,41.64750000000001, 0), v100, z5, tool0;
MoveL Offs(p0,118.04080000000006,40.82000000000001, 0), v100, z5, tool0;
MoveL Offs(p0,118.56269999999998,39.692499999999995, 0), v100, z5, tool0;
MoveL Offs(p0,119.1464,38.34, 0), v100, z5, tool0;
MoveL Offs(p0,119.7625,36.8375, 0), v100, z5, tool0;
MoveL Offs(p0,120.3816,35.260000000000005, 0), v100, z5, tool0;
MoveL Offs(p0,120.9743,33.6825, 0), v100, z5, tool0;
MoveL Offs(p0,121.5112,32.18000000000001, 0), v100, z5, tool0;
MoveL Offs(p0,121.96290000000002,30.827499999999997, 0), v100, z5, tool0;
MoveL Offs(p0,122.3,29.7, 0), v100, z5, tool0;
MoveL Offs(p0,121.74480000000001,29.45120000000001, 0), v100, z5, tool0;
